KUKA KRL program: MyProgram_278().src

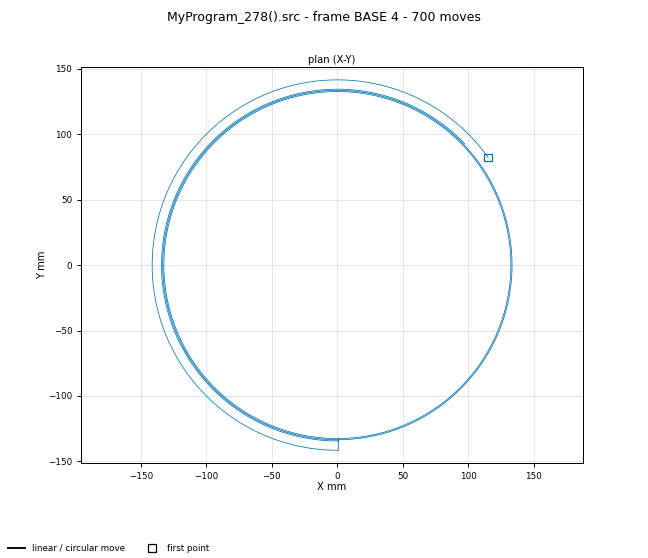
[picture p0: tool path of MyProgram_278().src in frame BASE 4, 700 of 700 moves have a stored position in this frame; points joined in program order, loops and branches not executed]
&ACCESS RVP
&REL 1
&PARAM TEMPLATE = C:\KRC\Roboter\Template\vorgabe
&PARAM EDITMASK = *
DEF MyProgram_278()
; ---- Setting reference (Base) ----
$BASE = BASE_DATA[4]

; --------------------------
; ---- Setting tool (TCP) ----
$TOOL = TOOL_DATA[3]
; --------------------------

$VEL.CP = VEL_APROX_PRINT
Startdeposition()
$VEL.CP = VEL_PRINT
LIN {X 115.1454,Y 82.1588,Z 172,A 37.1025,B 8.4652,C 0.1678,E1 8.5966,E2 414.6408} C_DIS
LIN {X 112.6327,Y 85.5722,Z 172,A 38.7723,B 8.4652,C 0.1649,E1 8.5938,E2 412.9763} C_DIS
LIN {X 109.941,Y 89.0032,Z 172,A 40.5158,B 8.4652,C 0.1614,E1 8.5908,E2 411.2351} C_DIS
LIN {X 107.1131,Y 92.3867,Z 172,A 42.2179,B 8.4653,C 0.1593,E1 8.5877,E2 409.5431} C_DIS
LIN {X 104.5819,Y 95.2429,Z 172,A 43.8363,B 8.4654,C 0.1545,E1 8.5847,E2 407.9148} C_DIS
LIN {X 101.4657,Y 98.556,Z 172,A 45.6031,B 8.4654,C 0.1523,E1 8.5813,E2 406.1572} C_DIS
LIN {X 98.3943,Y 101.6222,Z 172,A 47.3676,B 8.4655,C 0.1486,E1 8.5778,E2 404.3913} C_DIS
LIN {X 95.1433,Y 104.6723,Z 172,A 49.1662,B 8.4655,C 0.1453,E1 8.5741,E2 402.593} C_DIS
LIN {X 91.7276,Y 107.6782,Z 172,A 50.9618,B 8.4656,C 0.1428,E1 8.5703,E2 400.8031} C_DIS
LIN {X 88.3842,Y 110.4395,Z 172,A 52.7089,B 8.4656,C 0.1398,E1 8.5665,E2 399.0569} C_DIS
LIN {X 84.9572,Y 113.0968,Z 172,A 54.4403,B 8.4657,C 0.1373,E1 8.5627,E2 397.3283} C_DIS
LIN {X 81.4292,Y 115.6625,Z 172,A 56.2159,B 8.4657,C 0.1342,E1 8.5587,E2 395.5514} C_DIS
LIN {X 77.8557,Y 118.0975,Z 172,A 57.9483,B 8.4658,C 0.1318,E1 8.5546,E2 393.8213} C_DIS
LIN {X 74.2111,Y 120.4214,Z 172,A 59.7003,B 8.4658,C 0.1291,E1 8.5505,E2 392.069} C_DIS
LIN {X 70.4755,Y 122.6455,Z 172,A 61.4566,B 8.4658,C 0.1267,E1 8.5463,E2 390.3132} C_DIS
LIN {X 66.6565,Y 124.762,Z 172,A 63.2273,B 8.4659,C 0.1242,E1 8.5419,E2 388.5421} C_DIS
LIN {X 62.7995,Y 126.7448,Z 172,A 64.8378,B 8.4659,C 0.1249,E1 8.5379,E2 386.9504} C_DIS
LIN {X 59.6825,Y 128.2423,Z 172,A 66.2482,B 8.4659,C 0.123,E1 8.5344,E2 385.5388} C_DIS
LIN {X 56.3317,Y 129.7488,Z 172,A 67.58,B 8.4659,C 0.1245,E1 8.531,E2 384.2271} C_DIS
LIN {X 53.5262,Y 130.9328,Z 172,A 69.0454,B 8.4659,C 0.1185,E1 8.5272,E2 382.7321} C_DIS
LIN {X 49.8907,Y 132.3593,Z 172,A 70.6218,B 8.466,C 0.117,E1 8.5231,E2 381.1565} C_DIS
LIN {X 46.0135,Y 133.7567,Z 172,A 72.2511,B 8.466,C 0.1162,E1 8.5188,E2 379.5326} C_DIS
LIN {X 41.6859,Y 135.168,Z 172,A 73.8664,B 8.466,C 0.1192,E1 8.5146,E2 377.9469} C_DIS
LIN {X 38.5271,Y 136.1025,Z 172,A 75.2571,B 8.466,C 0.117,E1 8.5108,E2 376.5492} C_DIS
LIN {X 34.9773,Y 137.0571,Z 172,A 76.8136,B 8.466,C 0.1146,E1 8.5066,E2 374.9844} C_DIS
LIN {X 32.0331,Y 137.776,Z 172,A 78.0399,B 8.466,C 0.1138,E1 8.5033,E2 373.7585} C_DIS
LIN {X 28.648,Y 138.5191,Z 172,A 79.439,B 8.466,C 0.1131,E1 8.4994,E2 372.3604} C_DIS
LIN {X 25.2479,Y 139.1787,Z 172,A 80.6426,B 8.466,C 0.1162,E1 8.4962,E2 371.1827} C_DIS
LIN {X 22.4622,Y 139.6574,Z 172,A 81.9857,B 8.466,C 0.1119,E1 8.4924,E2 369.8146} C_DIS
LIN {X 19.0333,Y 140.165,Z 172,A 83.3905,B 8.466,C 0.1113,E1 8.4886,E2 368.4102} C_DIS
LIN {X 15.5815,Y 140.5898,Z 172,A 84.9056,B 8.4661,C 0.1088,E1 8.4843,E2 366.8819} C_DIS
LIN {X 11.0551,Y 141.0194,Z 172,A 86.7804,B 8.4661,C 0.1077,E1 8.4791,E2 365.0036} C_DIS
LIN {X 6.9219,Y 141.2807,Z 172,A 88.3854,B 8.4661,C 0.1089,E1 8.4746,E2 363.4085} C_DIS
LIN {X 2.8123,Y 141.4229,Z 172,A 89.8163,B 8.4661,C 0.1132,E1 8.4707,E2 362.0084} C_DIS
LIN {X -0.0523,Y 141.452,Z 172,A 91.1317,B 8.4661,C 0.1103,E1 8.467,E2 360.6737} C_DIS
LIN {X -3.4727,Y 141.4082,Z 172,A 92.5212,B 8.4661,C 0.1103,E1 8.4631,E2 359.2844} C_DIS
LIN {X -6.9499,Y 141.2793,Z 172,A 93.922,B 8.4661,C 0.1107,E1 8.4592,E2 357.8853} C_DIS
LIN {X -11.0634,Y 141.0188,Z 172,A 95.7118,B 8.4661,C 0.1088,E1 8.4542,E2 356.0811} C_DIS
LIN {X -15.5986,Y 140.588,Z 172,A 97.5605,B 8.4661,C 0.1093,E1 8.4491,E2 354.2329} C_DIS
LIN {X -20.8351,Y 139.9093,Z 172,A 99.5993,B 8.4661,C 0.112,E1 8.4435,E2 352.2082} C_DIS
LIN {X -24.2763,Y 139.3526,Z 172,A 101.0099,B 8.4661,C 0.1128,E1 8.4396,E2 350.7986} C_DIS
LIN {X -27.6797,Y 138.7161,Z 172,A 102.4085,B 8.4661,C 0.1136,E1 8.4357,E2 349.4013} C_DIS
LIN {X -31.0262,Y 138.0059,Z 172,A 103.7935,B 8.4661,C 0.1145,E1 8.432,E2 348.0172} C_DIS
LIN {X -34.3796,Y 137.2088,Z 172,A 105.204,B 8.4661,C 0.1152,E1 8.4281,E2 346.6058} C_DIS
LIN {X -37.7337,Y 136.3243,Z 172,A 106.6143,B 8.4661,C 0.1162,E1 8.4243,E2 345.1958} C_DIS
LIN {X -41.0644,Y 135.3582,Z 172,A 108.0256,B 8.4661,C 0.1173,E1 8.4206,E2 343.7846} C_DIS
LIN {X -44.3704,Y 134.3107,Z 172,A 109.5601,B 8.4661,C 0.1162,E1 8.4164,E2 342.2345} C_DIS
LIN {X -48.2905,Y 132.9516,Z 172,A 111.1286,B 8.466,C 0.1199,E1 8.4124,E2 340.6816} C_DIS
LIN {X -51.531,Y 131.7294,Z 172,A 112.5826,B 8.466,C 0.1205,E1 8.4086,E2 339.2221} C_DIS
LIN {X -55.7331,Y 130.0076,Z 172,A 114.4641,B 8.466,C 0.1218,E1 8.4037,E2 337.3366} C_DIS
LIN {X -59.1861,Y 128.4718,Z 172,A 115.8479,B 8.4659,C 0.1262,E1 8.4002,E2 335.9728} C_DIS
LIN {X -62.0494,Y 127.1148,Z 172,A 117.3081,B 8.4659,C 0.1248,E1 8.3965,E2 334.4911} C_DIS
LIN {X -65.4353,Y 125.4046,Z 172,A 118.8296,B 8.4659,C 0.1271,E1 8.3927,E2 332.9728} C_DIS
LIN {X -69.4478,Y 123.2297,Z 172,A 120.6863,B 8.4659,C 0.1296,E1 8.3882,E2 331.1167} C_DIS
LIN {X -73.1872,Y 121.0461,Z 172,A 122.4642,B 8.4659,C 0.1318,E1 8.3839,E2 329.3372} C_DIS
LIN {X -76.6775,Y 118.8666,Z 172,A 124.2067,B 8.4658,C 0.1331,E1 8.3798,E2 327.5865} C_DIS
LIN {X -80.4753,Y 116.3288,Z 172,A 126.0453,B 8.4658,C 0.1364,E1 8.3756,E2 325.751} C_DIS
LIN {X -84.0458,Y 113.776,Z 172,A 127.823,B 8.4657,C 0.1394,E1 8.3715,E2 323.9749} C_DIS
LIN {X -87.4843,Y 111.1532,Z 172,A 129.5764,B 8.4657,C 0.1425,E1 8.3677,E2 322.2229} C_DIS
LIN {X -90.7455,Y 108.5073,Z 172,A 131.3387,B 8.4656,C 0.1447,E1 8.3639,E2 320.4543} C_DIS
LIN {X -94.1347,Y 105.5807,Z 172,A 133.2066,B 8.4656,C 0.1473,E1 8.3599,E2 318.5812} C_DIS
LIN {X -97.5578,Y 102.4259,Z 172,A 135.0917,B 8.4655,C 0.151,E1 8.3561,E2 316.6979} C_DIS
LIN {X -100.7312,Y 99.307,Z 172,A 136.8846,B 8.4655,C 0.1549,E1 8.3526,E2 314.908} C_DIS
LIN {X -103.7389,Y 96.1607,Z 172,A 138.665,B 8.4654,C 0.1584,E1 8.3491,E2 313.127} C_DIS
LIN {X -106.7016,Y 92.8618,Z 172,A 140.4368,B 8.4653,C 0.1627,E1 8.3459,E2 311.3601} C_DIS
LIN {X -109.1769,Y 89.9391,Z 172,A 142.0776,B 8.4653,C 0.1647,E1 8.3429,E2 309.7093} C_DIS
LIN {X -111.717,Y 86.7632,Z 172,A 143.7599,B 8.4652,C 0.1679,E1 8.34,E2 308.0243} C_DIS
LIN {X -114.3228,Y 83.3004,Z 172,A 145.5562,B 8.4651,C 0.1714,E1 8.337,E2 306.2244} C_DIS
LIN {X -116.9427,Y 79.5804,Z 172,A 147.3892,B 8.4651,C 0.1759,E1 8.3341,E2 304.3946} C_DIS
LIN {X -119.3425,Y 75.9344,Z 172,A 149.1792,B 8.4649,C 0.1799,E1 8.3314,E2 302.6036} C_DIS
LIN {X -121.6068,Y 72.252,Z 172,A 150.9376,B 8.4649,C 0.1842,E1 8.3289,E2 300.846} C_DIS
LIN {X -123.7662,Y 68.487,Z 172,A 152.7274,B 8.4647,C 0.1881,E1 8.3264,E2 299.0539} C_DIS
LIN {X -125.8053,Y 64.6628,Z 172,A 154.5384,B 8.4647,C 0.1917,E1 8.3241,E2 297.2375} C_DIS
LIN {X -127.4923,Y 61.2682,Z 172,A 156.0158,B 8.4646,C 0.1967,E1 8.3223,E2 295.769} C_DIS
LIN {X -128.9555,Y 58.1258,Z 172,A 157.4972,B 8.4645,C 0.1992,E1 8.3205,E2 294.2791} C_DIS
LIN {X -130.4649,Y 54.6526,Z 172,A 158.986,B 8.4644,C 0.204,E1 8.3189,E2 292.7977} C_DIS
LIN {X -131.9767,Y 50.8947,Z 172,A 160.6744,B 8.4643,C 0.2077,E1 8.3172,E2 291.1048} C_DIS
LIN {X -133.1844,Y 47.6449,Z 172,A 162.1014,B 8.4643,C 0.2112,E1 8.3158,E2 289.6764} C_DIS
LIN {X -134.5157,Y 43.7501,Z 172,A 163.9142,B 8.4642,C 0.2134,E1 8.3142,E2 287.8465} C_DIS
LIN {X -135.5481,Y 40.4382,Z 172,A 165.2286,B 8.464,C 0.2188,E1 8.3131,E2 286.5452} C_DIS
LIN {X -136.4988,Y 37.1021,Z 172,A 166.7684,B 8.464,C 0.2206,E1 8.312,E2 284.9894} C_DIS
LIN {X -137.4708,Y 33.3144,Z 172,A 168.1472,B 8.4638,C 0.2283,E1 8.3111,E2 283.6387} C_DIS
LIN {X -138.1673,Y 30.2994,Z 172,A 169.5473,B 8.4638,C 0.2295,E1 8.3102,E2 282.2208} C_DIS
LIN {X -138.8695,Y 26.8965,Z 172,A 170.9776,B 8.4636,C 0.2332,E1 8.3094,E2 280.789} C_DIS
LIN {X -139.3798,Y 24.1242,Z 172,A 172.1369,B 8.4636,C 0.2362,E1 8.3088,E2 279.6286} C_DIS
LIN {X -139.9662,Y 20.4381,Z 172,A 173.5906,B 8.4634,C 0.2414,E1 8.3082,E2 278.1838} C_DIS
LIN {X -140.3869,Y 17.3177,Z 172,A 174.9932,B 8.4634,C 0.2431,E1 8.3077,E2 276.766} C_DIS
LIN {X -140.8329,Y 13.2018,Z 172,A 176.7152,B 8.4632,C 0.2472,E1 8.3072,E2 275.0397} C_DIS
LIN {X -141.1449,Y 9.3056,Z 172,A 178.1959,B 8.4631,C 0.2534,E1 8.3069,E2 273.5738} C_DIS
LIN {X -141.3295,Y 5.8467,Z 172,A 179.5992,B 8.4629,C 0.2574,E1 8.3067,E2 272.1718} C_DIS
LIN {X -141.4227,Y 2.8208,Z 172,A -178.9623,B 8.4629,C 0.2576,E1 8.3067,E2 270.7069} C_DIS
LIN {X -141.4499,Y -0.6582,Z 172,A -177.504,B 8.4629,C 0.2609,E1 8.3067,E2 269.2435} C_DIS
LIN {X -141.3775,Y -4.5742,Z 172,A -175.8333,B 8.4627,C 0.2641,E1 8.3067,E2 267.5633} C_DIS
LIN {X -141.1829,Y -8.6883,Z 172,A -174.2143,B 8.4626,C 0.2697,E1 8.307,E2 265.9522} C_DIS
LIN {X -140.8327,Y -13.2038,Z 172,A -172.3102,B 8.4624,C 0.2739,E1 8.3075,E2 264.0406} C_DIS
LIN {X -140.309,Y -17.9345,Z 172,A -170.4432,B 8.4622,C 0.2804,E1 8.3081,E2 262.1832} C_DIS
LIN {X -139.9212,Y -20.753,Z 172,A -169.2957,B 8.4621,C 0.2838,E1 8.3085,E2 261.0374} C_DIS
LIN {X -139.2931,Y -24.6084,Z 172,A -167.8031,B 8.4619,C 0.2897,E1 8.3092,E2 259.5577} C_DIS
LIN {X -138.7327,Y -27.598,Z 172,A -166.4153,B 8.4619,C 0.2907,E1 8.31,E2 258.1506} C_DIS
LIN {X -138.0138,Y -30.992,Z 172,A -164.988,B 8.4617,C 0.2943,E1 8.3108,E2 256.7216} C_DIS
LIN {X -137.0516,Y -34.9988,Z 172,A -163.2494,B 8.4617,C 0.2978,E1 8.312,E2 254.9751} C_DIS
LIN {X -135.8511,Y -39.4033,Z 172,A -161.4136,B 8.4614,C 0.3031,E1 8.3134,E2 253.1425} C_DIS
LIN {X -134.8446,Y -42.7206,Z 172,A -159.9867,B 8.4614,C 0.3066,E1 8.3146,E2 251.7137} C_DIS
LIN {X -133.5397,Y -46.6396,Z 172,A -158.2855,B 8.4612,C 0.3107,E1 8.3161,E2 250.01} C_DIS
LIN {X -132.2449,Y -50.1963,Z 172,A -156.5727,B 8.4612,C 0.3119,E1 8.3178,E2 248.2747} C_DIS
LIN {X -130.6879,Y -54.1187,Z 172,A -154.9897,B 8.4609,C 0.3185,E1 8.3194,E2 246.7094} C_DIS
LIN {X -129.3124,Y -57.3278,Z 172,A -153.5572,B 8.4607,C 0.3219,E1 8.321,E2 245.2756} C_DIS
LIN {X -127.8683,Y -60.481,Z 172,A -152.1318,B 8.4607,C 0.3251,E1 8.3227,E2 243.8483} C_DIS
LIN {X -126.1996,Y -63.8883,Z 172,A -150.5694,B 8.4605,C 0.3286,E1 8.3247,E2 242.2835} C_DIS
LIN {X -124.5929,Y -66.9712,Z 172,A -149.0497,B 8.4605,C 0.3303,E1 8.3267,E2 240.75} C_DIS
LIN {X -122.3755,Y -70.9421,Z 172,A -147.2166,B 8.4602,C 0.335,E1 8.3292,E2 238.9191} C_DIS
LIN {X -120.1302,Y -74.6812,Z 172,A -145.3688,B 8.4602,C 0.3379,E1 8.3319,E2 237.0616} C_DIS
LIN {X -117.6102,Y -78.59,Z 172,A -143.475,B 8.46,C 0.3422,E1 8.3348,E2 235.1675} C_DIS
LIN {X -115.1466,Y -82.1572,Z 172,A -141.6889,B 8.4598,C 0.3458,E1 8.3377,E2 233.3782} C_DIS
LIN {X -112.5749,Y -85.6478,Z 172,A -139.8928,B 8.4597,C 0.3491,E1 8.3407,E2 231.5777} C_DIS
LIN {X -109.8972,Y -89.0575,Z 172,A -138.0888,B 8.4595,C 0.3521,E1 8.3439,E2 229.7681} C_DIS
LIN {X -107.0913,Y -92.412,Z 172,A -136.3373,B 8.4594,C 0.3562,E1 8.347,E2 228.0199} C_DIS
LIN {X -103.996,Y -95.8822,Z 172,A -134.4237,B 8.4592,C 0.3596,E1 8.3506,E2 226.103} C_DIS
LIN {X -100.8648,Y -99.1708,Z 172,A -132.6103,B 8.4591,C 0.3638,E1 8.3541,E2 224.2937} C_DIS
LIN {X -97.94,Y -102.0605,Z 172,A -130.8665,B 8.459,C 0.3656,E1 8.3576,E2 222.54} C_DIS
LIN {X -94.52,Y -105.2356,Z 172,A -128.9605,B 8.4588,C 0.3689,E1 8.3616,E2 220.6324} C_DIS
LIN {X -91.0669,Y -108.2376,Z 172,A -127.1242,B 8.4587,C 0.3725,E1 8.3655,E2 218.7988} C_DIS
LIN {X -87.7072,Y -110.9782,Z 172,A -125.3297,B 8.4586,C 0.3749,E1 8.3694,E2 216.9996} C_DIS
LIN {X -84.2255,Y -113.6428,Z 172,A -123.5646,B 8.4584,C 0.378,E1 8.3733,E2 215.2362} C_DIS
LIN {X -80.7198,Y -116.1587,Z 172,A -121.8052,B 8.4584,C 0.3806,E1 8.3773,E2 213.4756} C_DIS
LIN {X -77.1326,Y -118.5711,Z 172,A -120.0273,B 8.4582,C 0.3827,E1 8.3815,E2 211.6943} C_DIS
LIN {X -73.4638,Y -120.8789,Z 172,A -118.2109,B 8.4582,C 0.3841,E1 8.3858,E2 209.87} C_DIS
LIN {X -69.6952,Y -123.0906,Z 172,A -116.4181,B 8.4581,C 0.3861,E1 8.3902,E2 208.0743} C_DIS
LIN {X -66.1771,Y -125.0151,Z 172,A -114.9013,B 8.4579,C 0.3901,E1 8.3939,E2 206.5717} C_DIS
LIN {X -62.808,Y -126.7406,Z 172,A -113.3542,B 8.4579,C 0.3917,E1 8.3977,E2 205.0228} C_DIS
LIN {X -59.6948,Y -128.2366,Z 172,A -111.9411,B 8.4578,C 0.393,E1 8.4013,E2 203.6078} C_DIS
LIN {X -56.3261,Y -129.7512,Z 172,A -110.5695,B 8.4576,C 0.3969,E1 8.4048,E2 202.2527} C_DIS
LIN {X -53.5252,Y -130.9332,Z 172,A -109.0853,B 8.4577,C 0.3935,E1 8.4087,E2 200.7348} C_DIS
LIN {X -49.2821,Y -132.5873,Z 172,A -107.3405,B 8.4576,C 0.397,E1 8.4132,E2 199.003} C_DIS
LIN {X -46.0166,Y -133.7557,Z 172,A -105.8454,B 8.4576,C 0.3965,E1 8.4172,E2 197.4957} C_DIS
LIN {X -41.4783,Y -135.2315,Z 172,A -104.0928,B 8.4574,C 0.4014,E1 8.4218,E2 195.7668} C_DIS
LIN {X -38.7552,Y -136.0387,Z 172,A -102.8288,B 8.4574,C 0.4,E1 8.4252,E2 194.4875} C_DIS
LIN {X -34.9861,Y -137.0549,Z 172,A -101.1431,B 8.4574,C 0.399,E1 8.4298,E2 192.7875} C_DIS
LIN {X -30.3504,Y -138.1563,Z 172,A -99.304,B 8.4574,C 0.4018,E1 8.4348,E2 190.96} C_DIS
LIN {X -26.9573,Y -138.8579,Z 172,A -97.8943,B 8.4574,C 0.4023,E1 8.4386,E2 189.5491} C_DIS
LIN {X -24.1772,Y -139.3703,Z 172,A -96.7641,B 8.4573,C 0.403,E1 8.4417,E2 188.4206} C_DIS
LIN {X -20.7465,Y -139.9221,Z 172,A -95.3306,B 8.4573,C 0.403,E1 8.4457,E2 186.9832} C_DIS
LIN {X -17.0562,Y -140.4181,Z 172,A -93.7579,B 8.4573,C 0.4021,E1 8.4501,E2 185.4013} C_DIS
LIN {X -13.2156,Y -140.8316,Z 172,A -92.2298,B 8.4573,C 0.4031,E1 8.4543,E2 183.8775} C_DIS
LIN {X -8.6601,Y -141.1847,Z 172,A -90.418,B 8.4573,C 0.404,E1 8.4594,E2 182.0701} C_DIS
LIN {X -4.5508,Y -141.3782,Z 172,A -88.7312,B 8.4573,C 0.4036,E1 8.4641,E2 180.3799} C_DIS
LIN {X -1.7323,Y -141.4408,Z 172,A -87.6287,B 8.4573,C 0.4043,E1 8.4671,E2 179.2822} C_DIS
LIN {X 1.0226,Y -141.4455,Z 172,A -86.8342,B 8.4569,C 0.4104,E1 8.4692,E2 178.5298} C_DIS
Enddeposition()
LIN {X 0.9597,Y -132.5053,Z 173,A -87.2924,B 8.5827,C 0.3662,E1 8.5925,E2 178.6674} C_DIS
Startdeposition()
$VEL.CP = VEL_PRINT
LIN {X -2.381,Y -132.4898,Z 173,A -88.9158,B 8.5825,C 0.3696,E1 8.5879,E2 180.3133} C_DIS
LIN {X -5.7833,Y -132.3862,Z 173,A -90.3521,B 8.5825,C 0.369,E1 8.5839,E2 181.7461} C_DIS
LIN {X -8.7494,Y -132.2232,Z 173,A -91.7266,B 8.5825,C 0.3706,E1 8.58,E2 183.1321} C_DIS
LIN {X -12.1019,Y -131.9584,Z 173,A -93.3007,B 8.5825,C 0.3725,E1 8.5756,E2 184.7214} C_DIS
LIN {X -16.2246,Y -131.5149,Z 173,A -94.9013,B 8.5825,C 0.3687,E1 8.5712,E2 186.2992} C_DIS
LIN {X -19.4498,Y -131.0776,Z 173,A -96.3155,B 8.5825,C 0.3684,E1 8.5673,E2 187.7147} C_DIS
LIN {X -22.6582,Y -130.5611,Z 173,A -97.7413,B 8.5825,C 0.3684,E1 8.5634,E2 189.1435} C_DIS
LIN {X -25.8503,Y -129.9662,Z 173,A -99.1463,B 8.5826,C 0.3677,E1 8.5595,E2 190.549} C_DIS
LIN {X -29.7453,Y -129.1293,Z 173,A -100.8844,B 8.5826,C 0.3671,E1 8.5548,E2 192.2894} C_DIS
LIN {X -33.7754,Y -128.1345,Z 173,A -102.6831,B 8.5826,C 0.3661,E1 8.5499,E2 194.089} C_DIS
LIN {X -36.9449,Y -127.2566,Z 173,A -104.0949,B 8.5827,C 0.365,E1 8.5461,E2 195.4998} C_DIS
LIN {X -40.4074,Y -126.1995,Z 173,A -105.7344,B 8.5827,C 0.365,E1 8.5417,E2 197.1486} C_DIS
LIN {X -43.8059,Y -125.0611,Z 173,A -107.226,B 8.5828,C 0.3628,E1 8.5378,E2 198.6334} C_DIS
LIN {X -47.0117,Y -123.8922,Z 173,A -108.8671,B 8.5828,C 0.3643,E1 8.5334,E2 200.2948} C_DIS
LIN {X -51.1864,Y -122.2253,Z 173,A -110.7174,B 8.5829,C 0.3608,E1 8.5287,E2 202.1339} C_DIS
LIN {X -54.5147,Y -120.7782,Z 173,A -112.3809,B 8.5829,C 0.3608,E1 8.5244,E2 203.809} C_DIS
LIN {X -58.1203,Y -119.0855,Z 173,A -113.9715,B 8.5831,C 0.3566,E1 8.5204,E2 205.3837} C_DIS
LIN {X -61.0215,Y -117.6258,Z 173,A -115.369,B 8.5831,C 0.3547,E1 8.517,E2 206.7803} C_DIS
LIN {X -63.9076,Y -116.084,Z 173,A -116.9596,B 8.5831,C 0.3559,E1 8.513,E2 208.3922} C_DIS
LIN {X -67.5035,Y -114.0307,Z 173,A -118.6243,B 8.5833,C 0.3514,E1 8.509,E2 210.0417} C_DIS
LIN {X -70.2751,Y -112.3435,Z 173,A -120.0427,B 8.5833,C 0.3496,E1 8.5056,E2 211.4618} C_DIS
LIN {X -73.6197,Y -110.1803,Z 173,A -121.818,B 8.5834,C 0.3479,E1 8.5015,E2 213.2434} C_DIS
LIN {X -77.0465,Y -107.8119,Z 173,A -123.5913,B 8.5836,C 0.3446,E1 8.4974,E2 215.013} C_DIS
LIN {X -79.6565,Y -105.8982,Z 173,A -125.1381,B 8.5836,C 0.3447,E1 8.4939,E2 216.5774} C_DIS
LIN {X -83.0306,Y -103.274,Z 173,A -126.9759,B 8.5836,C 0.3414,E1 8.4899,E2 218.4136} C_DIS
LIN {X -86.277,Y -100.5778,Z 173,A -128.7973,B 8.5838,C 0.3381,E1 8.486,E2 220.2341} C_DIS
LIN {X -89.3334,Y -97.8737,Z 173,A -130.5836,B 8.5839,C 0.3352,E1 8.4823,E2 222.0226} C_DIS
LIN {X -92.2223,Y -95.1557,Z 173,A -132.3094,B 8.5841,C 0.3321,E1 8.4788,E2 223.7492} C_DIS
LIN {X -95.154,Y -92.224,Z 173,A -134.123,B 8.5841,C 0.3288,E1 8.4753,E2 225.5647} C_DIS
LIN {X -97.9916,Y -89.2034,Z 173,A -135.9986,B 8.5843,C 0.3265,E1 8.4717,E2 227.4498} C_DIS
LIN {X -101.1067,Y -85.6565,Z 173,A -138.0254,B 8.5844,C 0.3219,E1 8.468,E2 229.474} C_DIS
LIN {X -103.7467,Y -82.439,Z 173,A -139.8152,B 8.5846,C 0.3178,E1 8.4649,E2 231.262} C_DIS
LIN {X -106.4386,Y -78.9332,Z 173,A -141.8433,B 8.5846,C 0.3153,E1 8.4614,E2 233.3032} C_DIS
LIN {X -108.7586,Y -75.7041,Z 173,A -143.506,B 8.5849,C 0.3105,E1 8.4587,E2 234.9583} C_DIS
LIN {X -111.0758,Y -72.2617,Z 173,A -145.2555,B 8.585,C 0.3056,E1 8.4561,E2 236.7016} C_DIS
LIN {X -113.1978,Y -68.8909,Z 173,A -147.0175,B 8.5852,C 0.302,E1 8.4535,E2 238.4675} C_DIS
LIN {X -114.9544,Y -65.9177,Z 173,A -148.5138,B 8.5852,C 0.2984,E1 8.4513,E2 239.9633} C_DIS
LIN {X -116.8718,Y -62.4551,Z 173,A -150.2717,B 8.5854,C 0.2949,E1 8.449,E2 241.7258} C_DIS
LIN {X -118.3626,Y -59.5793,Z 173,A -151.6868,B 8.5855,C 0.2915,E1 8.4472,E2 243.1417} C_DIS
LIN {X -119.7842,Y -56.6659,Z 173,A -153.1098,B 8.5856,C 0.2883,E1 8.4455,E2 244.5665} C_DIS
LIN {X -121.1428,Y -53.6996,Z 173,A -154.5405,B 8.5857,C 0.2849,E1 8.4438,E2 245.9987} C_DIS
LIN {X -122.4234,Y -50.712,Z 173,A -155.9674,B 8.5858,C 0.2815,E1 8.4423,E2 247.4271} C_DIS
LIN {X -123.9001,Y -46.9905,Z 173,A -157.769,B 8.586,C 0.2779,E1 8.4404,E2 249.236} C_DIS
LIN {X -125.3043,Y -43.1044,Z 173,A -159.5681,B 8.5861,C 0.2733,E1 8.4388,E2 251.0353} C_DIS
LIN {X -126.5848,Y -39.1859,Z 173,A -161.3934,B 8.5862,C 0.2691,E1 8.4372,E2 252.8644} C_DIS
LIN {X -127.5391,Y -35.9575,Z 173,A -162.9581,B 8.5863,C 0.2667,E1 8.436,E2 254.4411} C_DIS
LIN {X -128.7239,Y -31.455,Z 173,A -164.92,B 8.5865,C 0.2603,E1 8.4346,E2 256.3953} C_DIS
LIN {X -129.4826,Y -28.1674,Z 173,A -166.4827,B 8.5865,C 0.2578,E1 8.4337,E2 257.9692} C_DIS
LIN {X -130.2665,Y -24.2924,Z 173,A -168.0949,B 8.5868,C 0.2515,E1 8.4328,E2 259.5685} C_DIS
LIN {X -130.8301,Y -21.0524,Z 173,A -169.5586,B 8.5868,C 0.2481,E1 8.4321,E2 261.036} C_DIS
LIN {X -131.3061,Y -17.8395,Z 173,A -170.9918,B 8.587,C 0.2445,E1 8.4316,E2 262.4715} C_DIS
LIN {X -131.687,Y -14.7654,Z 173,A -172.3999,B 8.587,C 0.2417,E1 8.4311,E2 263.8866} C_DIS
LIN {X -132.0225,Y -11.3691,Z 173,A -173.9578,B 8.5871,C 0.2386,E1 8.4307,E2 265.4529} C_DIS
LIN {X -132.3143,Y -7.2414,Z 173,A -175.6293,B 8.5873,C 0.2317,E1 8.4304,E2 267.109} C_DIS
LIN {X -132.4468,Y -4.1512,Z 173,A -177.0764,B 8.5873,C 0.2295,E1 8.4303,E2 268.5678} C_DIS
LIN {X -132.5145,Y 0.0019,Z 173,A -179.0708,B 8.5874,C 0.2272,E1 8.4303,E2 270.5841} C_DIS
LIN {X -132.4471,Y 4.1413,Z 173,A 179.3434,B 8.5877,C 0.219,E1 8.4303,E2 272.1441} C_DIS
LIN {X -132.3149,Y 7.2293,Z 173,A 177.943,B 8.5877,C 0.2161,E1 8.4305,E2 273.5508} C_DIS
LIN {X -132.0346,Y 11.2266,Z 173,A 176.1471,B 8.5878,C 0.212,E1 8.4309,E2 275.3525} C_DIS
LIN {X -131.6023,Y 15.4923,Z 173,A 174.1997,B 8.5879,C 0.208,E1 8.4315,E2 277.3092} C_DIS
LIN {X -131.0789,Y 19.4409,Z 173,A 172.5751,B 8.5881,C 0.2016,E1 8.4321,E2 278.9207} C_DIS
LIN {X -130.5949,Y 22.4616,Z 173,A 171.2403,B 8.5881,C 0.198,E1 8.4327,E2 280.2556} C_DIS
LIN {X -129.9526,Y 25.9171,Z 173,A 169.687,B 8.5882,C 0.1942,E1 8.4336,E2 281.8114} C_DIS
LIN {X -129.1237,Y 29.7699,Z 173,A 167.9225,B 8.5883,C 0.1902,E1 8.4346,E2 283.5813} C_DIS
LIN {X -128.133,Y 33.7809,Z 173,A 166.1187,B 8.5884,C 0.1854,E1 8.4359,E2 285.3854} C_DIS
LIN {X -127.06,Y 37.6163,Z 173,A 164.3416,B 8.5885,C 0.1814,E1 8.4372,E2 287.1672} C_DIS
LIN {X -125.8238,Y 41.5635,Z 173,A 162.5506,B 8.5886,C 0.1765,E1 8.4388,E2 288.9568} C_DIS
LIN {X -124.5199,Y 45.3211,Z 173,A 160.7496,B 8.5886,C 0.173,E1 8.4404,E2 290.7656} C_DIS
LIN {X -123.037,Y 49.2044,Z 173,A 158.904,B 8.5888,C 0.1688,E1 8.4423,E2 292.615} C_DIS
LIN {X -121.4322,Y 53.0424,Z 173,A 157.1426,B 8.5888,C 0.1634,E1 8.4442,E2 294.3702} C_DIS
LIN {X -119.7861,Y 56.6619,Z 173,A 155.405,B 8.589,C 0.1592,E1 8.4463,E2 296.1083} C_DIS
LIN {X -118.3617,Y 59.581,Z 173,A 153.9803,B 8.589,C 0.1558,E1 8.448,E2 297.534} C_DIS
LIN {X -116.867,Y 62.464,Z 173,A 152.5289,B 8.589,C 0.1529,E1 8.4499,E2 298.9895} C_DIS
LIN {X -114.8994,Y 66.0141,Z 173,A 150.7336,B 8.5891,C 0.149,E1 8.4524,E2 300.7878} C_DIS
LIN {X -113.1833,Y 68.9149,Z 173,A 149.2803,B 8.5892,C 0.1453,E1 8.4545,E2 302.2391} C_DIS
LIN {X -111.473,Y 71.6476,Z 173,A 147.868,B 8.5892,C 0.1421,E1 8.4566,E2 303.6522} C_DIS
LIN {X -109.2807,Y 74.9485,Z 173,A 145.9887,B 8.5892,C 0.1405,E1 8.4595,E2 305.5491} C_DIS
LIN {X -106.8723,Y 78.3446,Z 173,A 144.3089,B 8.5894,C 0.1344,E1 8.4623,E2 307.213} C_DIS
LIN {X -104.4711,Y 81.52,Z 173,A 142.4663,B 8.5894,C 0.1322,E1 8.4654,E2 309.0681} C_DIS
LIN {X -101.91,Y 84.6992,Z 173,A 140.684,B 8.5894,C 0.1285,E1 8.4686,E2 310.8507} C_DIS
LIN {X -99.0269,Y 88.0532,Z 173,A 138.7326,B 8.5895,C 0.1249,E1 8.4722,E2 312.8048} C_DIS
LIN {X -96.2776,Y 91.0505,Z 173,A 136.9714,B 8.5895,C 0.1212,E1 8.4755,E2 314.5646} C_DIS
LIN {X -93.3768,Y 94.023,Z 173,A 135.1693,B 8.5896,C 0.1175,E1 8.479,E2 316.3657} C_DIS
LIN {X -90.4564,Y 96.8361,Z 173,A 133.3818,B 8.5896,C 0.1145,E1 8.4827,E2 318.1556} C_DIS
LIN {X -87.4521,Y 99.5583,Z 173,A 131.5938,B 8.5897,C 0.1116,E1 8.4864,E2 319.946} C_DIS
LIN {X -84.3407,Y 102.2069,Z 173,A 129.8318,B 8.5897,C 0.1082,E1 8.4902,E2 321.7058} C_DIS
LIN {X -81.2337,Y 104.6931,Z 173,A 128.0528,B 8.5897,C 0.106,E1 8.4941,E2 323.49} C_DIS
LIN {X -78.6888,Y 106.6195,Z 173,A 126.6434,B 8.5898,C 0.1041,E1 8.4972,E2 324.9016} C_DIS
LIN {X -75.4206,Y 108.9559,Z 173,A 124.8966,B 8.5898,C 0.1013,E1 8.5012,E2 326.648} C_DIS
LIN {X -72.2432,Y 111.0878,Z 173,A 123.3388,B 8.5898,C 0.0971,E1 8.5048,E2 328.193} C_DIS
LIN {X -69.501,Y 112.8239,Z 173,A 121.7857,B 8.5898,C 0.0973,E1 8.5085,E2 329.7624} C_DIS
LIN {X -65.9466,Y 114.9379,Z 173,A 120.1216,B 8.5899,C 0.0927,E1 8.5125,E2 331.4105} C_DIS
LIN {X -62.4687,Y 116.8645,Z 173,A 118.3572,B 8.5899,C 0.091,E1 8.5169,E2 333.1788} C_DIS
LIN {X -59.5869,Y 118.3587,Z 173,A 116.9597,B 8.5899,C 0.089,E1 8.5203,E2 334.5744} C_DIS
LIN {X -56.6527,Y 119.7905,Z 173,A 115.5396,B 8.5899,C 0.0874,E1 8.5239,E2 335.9943} C_DIS
LIN {X -53.6996,Y 121.1428,Z 173,A 114.1226,B 8.59,C 0.0859,E1 8.5275,E2 337.4117} C_DIS
LIN {X -50.6793,Y 122.437,Z 173,A 112.6975,B 8.59,C 0.0843,E1 8.5312,E2 338.8362} C_DIS
LIN {X -47.6723,Y 123.6387,Z 173,A 111.2891,B 8.59,C 0.0829,E1 8.5348,E2 340.2445} C_DIS
LIN {X -44.6334,Y 124.7679,Z 173,A 109.7555,B 8.59,C 0.0837,E1 8.5389,E2 341.7925} C_DIS
LIN {X -40.8715,Y 126.0512,Z 173,A 108.1051,B 8.59,C 0.081,E1 8.5432,E2 343.4337} C_DIS
LIN {X -37.6298,Y 127.0561,Z 173,A 106.6764,B 8.59,C 0.0791,E1 8.5471,E2 344.8568} C_DIS
LIN {X -33.7713,Y 128.1356,Z 173,A 104.7966,B 8.59,C 0.0802,E1 8.5522,E2 346.7526} C_DIS
LIN {X -29.5409,Y 129.176,Z 173,A 102.9667,B 8.59,C 0.078,E1 8.5571,E2 348.575} C_DIS
LIN {X -25.8433,Y 129.9676,Z 173,A 101.4112,B 8.59,C 0.0757,E1 8.5613,E2 350.1203} C_DIS
LIN {X -22.6485,Y 130.5629,Z 173,A 100.0051,B 8.5901,C 0.0749,E1 8.5652,E2 351.5257} C_DIS
LIN {X -19.4417,Y 131.0788,Z 173,A 98.5726,B 8.5901,C 0.0748,E1 8.5692,E2 352.9606} C_DIS
LIN {X -16.2228,Y 131.5152,Z 173,A 97.164,B 8.5901,C 0.0743,E1 8.5731,E2 354.3688} C_DIS
LIN {X -12.9861,Y 131.8735,Z 173,A 95.7576,B 8.5901,C 0.0738,E1 8.577,E2 355.7743} C_DIS
LIN {X -9.4578,Y 132.1732,Z 173,A 94.1414,B 8.5901,C 0.0749,E1 8.5815,E2 357.3996} C_DIS
LIN {X -5.766,Y 132.3869,Z 173,A 92.6148,B 8.5901,C 0.0734,E1 8.5857,E2 358.917} C_DIS
LIN {X -2.2547,Y 132.4919,Z 173,A 91.0315,B 8.5901,C 0.0744,E1 8.5902,E2 360.5071} C_DIS
LIN {X 1.6374,Y 132.5022,Z 173,A 89.4118,B 8.5901,C 0.0733,E1 8.5947,E2 362.1187} C_DIS
LIN {X 4.8828,Y 132.4213,Z 173,A 88.0191,B 8.5901,C 0.0732,E1 8.5985,E2 363.5095} C_DIS
LIN {X 8.3922,Y 132.2452,Z 173,A 86.4048,B 8.5901,C 0.0751,E1 8.6031,E2 365.1342} C_DIS
LIN {X 12.0962,Y 131.9589,Z 173,A 84.8459,B 8.5901,C 0.0746,E1 8.6074,E2 366.6871} C_DIS
LIN {X 16.2274,Y 131.5146,Z 173,A 83.1228,B 8.5901,C 0.0739,E1 8.6122,E2 368.4009} C_DIS
LIN {X 19.4474,Y 131.078,Z 173,A 81.7178,B 8.5901,C 0.0744,E1 8.616,E2 369.8056} C_DIS
LIN {X 22.6549,Y 130.5617,Z 173,A 80.2978,B 8.5901,C 0.0753,E1 8.62,E2 371.2269} C_DIS
LIN {X 25.8477,Y 129.9667,Z 173,A 78.9007,B 8.5901,C 0.0759,E1 8.6238,E2 372.6227} C_DIS
LIN {X 29.755,Y 129.1271,Z 173,A 77.1616,B 8.5901,C 0.0772,E1 8.6285,E2 374.3627} C_DIS
LIN {X 33.8136,Y 128.1243,Z 173,A 75.3866,B 8.5901,C 0.0778,E1 8.6333,E2 376.1335} C_DIS
LIN {X 36.9278,Y 127.2616,Z 173,A 73.9955,B 8.5901,C 0.0788,E1 8.6371,E2 377.5236} C_DIS
LIN {X 40.8724,Y 126.051,Z 173,A 72.2206,B 8.5901,C 0.0802,E1 8.6418,E2 379.2971} C_DIS
LIN {X 44.646,Y 124.7633,Z 173,A 70.3505,B 8.5901,C 0.0845,E1 8.6468,E2 381.184} C_DIS
LIN {X 49.2064,Y 123.0362,Z 173,A 68.3019,B 8.5901,C 0.0855,E1 8.6521,E2 383.2254} C_DIS
LIN {X 53.0254,Y 121.4396,Z 173,A 66.6277,B 8.5901,C 0.0854,E1 8.6563,E2 384.886} C_DIS
LIN {X 56.6534,Y 119.7902,Z 173,A 64.9264,B 8.59,C 0.087,E1 8.6606,E2 386.5847} C_DIS
LIN {X 59.5734,Y 118.3656,Z 173,A 63.604,B 8.59,C 0.0872,E1 8.6639,E2 387.8974} C_DIS
LIN {X 62.4779,Y 116.8595,Z 173,A 62.1271,B 8.59,C 0.0903,E1 8.6676,E2 389.3817} C_DIS
LIN {X 65.9613,Y 114.9295,Z 173,A 60.3896,B 8.59,C 0.093,E1 8.6718,E2 391.1211} C_DIS
LIN {X 69.5154,Y 112.8151,Z 173,A 58.639,B 8.59,C 0.0949,E1 8.676,E2 392.8675} C_DIS
LIN {X 72.399,Y 110.9866,Z 173,A 57.0259,B 8.5899,C 0.0998,E1 8.6798,E2 394.4968} C_DIS
LIN {X 75.7245,Y 108.7445,Z 173,A 55.4111,B 8.5899,C 0.1003,E1 8.6835,E2 396.0977} C_DIS
LIN {X 78.9333,Y 106.4385,Z 173,A 53.6782,B 8.5899,C 0.1037,E1 8.6874,E2 397.8338} C_DIS
LIN {X 82.1697,Y 103.9608,Z 173,A 51.9435,B 8.5898,C 0.1062,E1 8.6913,E2 399.5656} C_DIS
LIN {X 85.3168,Y 101.3934,Z 173,A 50.1759,B 8.5898,C 0.1097,E1 8.6951,E2 401.335} C_DIS
LIN {X 88.6954,Y 98.4522,Z 173,A 48.2852,B 8.5897,C 0.1124,E1 8.699,E2 403.2207} C_DIS
LIN {X 91.641,Y 95.7158,Z 173,A 46.5831,B 8.5897,C 0.1151,E1 8.7025,E2 404.919} C_DIS
LIN {X 94.9019,Y 92.4844,Z 173,A 44.6063,B 8.5897,C 0.119,E1 8.7064,E2 406.8955} C_DIS
LIN {X 97.8877,Y 89.318,Z 173,A 42.7388,B 8.5896,C 0.1227,E1 8.7099,E2 408.762} C_DIS
LIN {X 100.637,Y 86.2083,Z 173,A 40.9771,B 8.5896,C 0.1259,E1 8.7131,E2 410.5205} C_DIS
LIN {X 103.2502,Y 83.0601,Z 173,A 39.2651,B 8.5895,C 0.1287,E1 8.7161,E2 412.2264} C_DIS
LIN {X 105.9051,Y 79.6474,Z 173,A 37.4149,B 8.5895,C 0.1325,E1 8.7193,E2 414.0751} C_DIS
LIN {X 108.3441,Y 76.2963,Z 173,A 35.7052,B 8.5894,C 0.135,E1 8.7221,E2 415.7759} C_DIS
LIN {X 110.1816,Y 73.6178,Z 173,A 34.3229,B 8.5894,C 0.1379,E1 8.7242,E2 417.1562} C_DIS
LIN {X 111.9531,Y 70.895,Z 173,A 32.9405,B 8.5893,C 0.1409,E1 8.7263,E2 418.5367} C_DIS
LIN {X 114.0319,Y 67.5014,Z 173,A 31.2081,B 8.5893,C 0.1453,E1 8.7288,E2 420.2714} C_DIS
LIN {X 115.7271,Y 64.552,Z 173,A 29.6438,B 8.5891,C 0.1509,E1 8.731,E2 421.8477} C_DIS
LIN {X 117.3482,Y 61.5501,Z 173,A 28.2565,B 8.5891,C 0.1528,E1 8.7328,E2 423.2253} C_DIS
LIN {X 119.0863,Y 58.1189,Z 173,A 26.6952,B 8.5891,C 0.155,E1 8.7347,E2 424.7756} C_DIS
LIN {X 120.4747,Y 55.1824,Z 173,A 25.3137,B 8.589,C 0.1582,E1 8.7363,E2 426.1552} C_DIS
LIN {X 121.7437,Y 52.322,Z 173,A 23.9687,B 8.589,C 0.1616,E1 8.7378,E2 427.5001} C_DIS
LIN {X 123.0479,Y 49.1774,Z 173,A 22.4078,B 8.5888,C 0.1674,E1 8.7395,E2 429.0726} C_DIS
LIN {X 124.7672,Y 44.6352,Z 173,A 20.47,B 8.5888,C 0.1697,E1 8.7413,E2 430.9925} C_DIS
LIN {X 125.8213,Y 41.571,Z 173,A 19.0922,B 8.5887,C 0.173,E1 8.7426,E2 432.3685} C_DIS
LIN {X 126.9564,Y 37.9701,Z 173,A 17.3724,B 8.5886,C 0.1794,E1 8.744,E2 434.1} C_DIS
LIN {X 127.9453,Y 34.4847,Z 173,A 15.9422,B 8.5886,C 0.1809,E1 8.7451,E2 435.5151} C_DIS
LIN {X 128.7534,Y 31.3325,Z 173,A 14.4324,B 8.5884,C 0.1869,E1 8.7461,E2 437.0382} C_DIS
LIN {X 129.639,Y 27.4432,Z 173,A 12.8703,B 8.5884,C 0.1884,E1 8.747,E2 438.5822} C_DIS
LIN {X 130.2736,Y 24.2553,Z 173,A 11.4916,B 8.5883,C 0.1918,E1 8.7477,E2 439.9588} C_DIS
LIN {X 130.8297,Y 21.0545,Z 173,A 10.115,B 8.5883,C 0.1953,E1 8.7484,E2 441.3333} C_DIS
LIN {X 131.3081,Y 17.8241,Z 173,A 8.7008,B 8.5881,C 0.1993,E1 8.7489,E2 442.7489} C_DIS
LIN {X 131.7047,Y 14.6014,Z 173,A 7.174,B 8.588,C 0.2059,E1 8.7494,E2 444.2916} C_DIS
LIN {X 132.0843,Y 10.6376,Z 173,A 5.6553,B 8.588,C 0.2066,E1 8.7498,E2 445.7874} C_DIS
LIN {X 132.3142,Y 7.2437,Z 173,A 4.2179,B 8.5879,C 0.2102,E1 8.75,E2 447.2221} C_DIS
LIN {X 132.4474,Y 4.1308,Z 173,A 2.8212,B 8.5878,C 0.2151,E1 8.7502,E2 448.626} C_DIS
LIN {X 132.5145,Y -0.0034,Z 173,A 0.9018,B 8.5876,C 0.2231,E1 8.7502,E2 450.5629} C_DIS
LIN {X 132.4472,Y -4.1388,Z 173,A -0.6298,B 8.5876,C 0.2228,E1 8.7502,E2 452.0651} C_DIS
LIN {X 132.3265,Y -6.9997,Z 173,A -1.912,B 8.5874,C 0.2274,E1 8.75,E2 453.3538} C_DIS
LIN {X 132.0915,Y -10.5521,Z 173,A -3.3716,B 8.5874,C 0.2301,E1 8.7497,E2 454.8053} C_DIS
LIN {X 131.7853,Y -13.8521,Z 173,A -4.7988,B 8.5873,C 0.2342,E1 8.7493,E2 456.2331} C_DIS
LIN {X 131.3072,Y -17.831,Z 173,A -6.4768,B 8.5872,C 0.238,E1 8.7487,E2 457.9062} C_DIS
LIN {X 130.8319,Y -21.0414,Z 173,A -7.8554,B 8.5871,C 0.2415,E1 8.7481,E2 459.2833} C_DIS
LIN {X 130.1349,Y -24.9805,Z 173,A -9.5679,B 8.5869,C 0.2461,E1 8.7472,E2 460.9953} C_DIS
LIN {X 129.442,Y -28.3554,Z 173,A -11.1838,B 8.5867,C 0.253,E1 8.7463,E2 462.628} C_DIS
LIN {X 128.5264,Y -32.252,Z 173,A -12.872,B 8.5867,C 0.257,E1 8.7452,E2 464.3127} C_DIS
LIN {X 127.2828,Y -36.8554,Z 173,A -14.9135,B 8.5864,C 0.2624,E1 8.7436,E2 466.3538} C_DIS
LIN {X 125.9448,Y -41.2002,Z 173,A -16.8095,B 8.5864,C 0.2664,E1 8.742,E2 468.2434} C_DIS
LIN {X 124.5129,Y -45.3406,Z 173,A -18.576,B 8.5862,C 0.269,E1 8.7404,E2 469.9963} C_DIS
LIN {X 123.0368,Y -49.2049,Z 173,A -20.393,B 8.5861,C 0.2745,E1 8.7386,E2 471.8186} C_DIS
LIN {X 121.4128,Y -53.0873,Z 173,A -22.1152,B 8.586,C 0.2773,E1 8.7367,E2 473.5309} C_DIS
LIN {X 120.1518,Y -55.8807,Z 173,A -23.418,B 8.5859,C 0.2804,E1 8.7352,E2 474.8323} C_DIS
LIN {X 118.4682,Y -59.3719,Z 173,A -25.1395,B 8.5857,C 0.2858,E1 8.733,E2 476.5611} C_DIS
LIN {X 116.8681,Y -62.4619,Z 173,A -26.5418,B 8.5857,C 0.2876,E1 8.7312,E2 477.9525} C_DIS
LIN {X 114.9503,Y -65.9249,Z 173,A -28.2622,B 8.5855,C 0.2922,E1 8.7289,E2 479.6757} C_DIS
LIN {X 113.2023,Y -68.8836,Z 173,A -29.8448,B 8.5853,C 0.2979,E1 8.7266,E2 481.2716} C_DIS
LIN {X 110.7799,Y -72.7145,Z 173,A -31.7021,B 8.5853,C 0.3007,E1 8.7238,E2 483.1184} C_DIS
LIN {X 108.8022,Y -75.6415,Z 173,A -33.1491,B 8.5851,C 0.3028,E1 8.7215,E2 484.5573} C_DIS
LIN {X 106.8711,Y -78.3462,Z 173,A -34.5455,B 8.5851,C 0.3054,E1 8.7192,E2 485.9502} C_DIS
LIN {X 104.9621,Y -80.8867,Z 173,A -35.9877,B 8.5849,C 0.3101,E1 8.7168,E2 487.4021} C_DIS
LIN {X 102.3196,Y -84.2047,Z 173,A -37.7965,B 8.5847,C 0.3138,E1 8.7136,E2 489.2097} C_DIS
LIN {X 99.5407,Y -87.4721,Z 173,A -39.635,B 8.5846,C 0.3176,E1 8.7103,E2 491.048} C_DIS
LIN {X 96.8313,Y -90.4616,Z 173,A -41.3469,B 8.5845,C 0.3208,E1 8.707,E2 492.7577} C_DIS
LIN {X 94.0148,Y -93.3851,Z 173,A -43.1064,B 8.5843,C 0.3247,E1 8.7036,E2 494.5194} C_DIS
LIN {X 90.9932,Y -96.3317,Z 173,A -44.8594,B 8.5843,C 0.327,E1 8.7001,E2 496.2654} C_DIS
LIN {X 88.0485,Y -99.0311,Z 173,A -46.5906,B 8.5841,C 0.3306,E1 8.6965,E2 497.9988} C_DIS
LIN {X 84.9737,Y -101.6814,Z 173,A -48.318,B 8.584,C 0.3335,E1 8.6928,E2 499.7245} C_DIS
LIN {X 81.7995,Y -104.2516,Z 173,A -50.0471,B 8.5839,C 0.3361,E1 8.689,E2 501.4507} C_DIS
LIN {X 78.348,Y -106.8698,Z 173,A -51.9757,B 8.5837,C 0.3406,E1 8.6847,E2 503.3879} C_DIS
LIN {X 74.9651,Y -109.2694,Z 173,A -53.763,B 8.5837,C 0.3436,E1 8.6806,E2 505.1761} C_DIS
LIN {X 70.9752,Y -111.9025,Z 173,A -55.7074,B 8.5836,C 0.3446,E1 8.6761,E2 507.1074} C_DIS
LIN {X 67.4216,Y -114.079,Z 173,A -57.4779,B 8.5835,C 0.3469,E1 8.6719,E2 508.8756} C_DIS
LIN {X 64.5322,Y -115.7381,Z 173,A -59.0217,B 8.5833,C 0.3511,E1 8.6681,E2 510.4333} C_DIS
LIN {X 61.0316,Y -117.6205,Z 173,A -60.588,B 8.5833,C 0.3506,E1 8.6642,E2 511.9824} C_DIS
LIN {X 58.1127,Y -119.0893,Z 173,A -61.9865,B 8.5833,C 0.3523,E1 8.6607,E2 513.3803} C_DIS
LIN {X 55.1766,Y -120.4774,Z 173,A -63.5155,B 8.5831,C 0.3566,E1 8.6568,E2 514.9256} C_DIS
LIN {X 50.9423,Y -122.3272,Z 173,A -65.3941,B 8.5831,C 0.3568,E1 8.652,E2 516.7913} C_DIS
LIN {X 47.01,Y -123.8928,Z 173,A -67.2197,B 8.583,C 0.3588,E1 8.6473,E2 518.6178} C_DIS
LIN {X 43.21,Y -125.2677,Z 173,A -68.9409,B 8.583,C 0.3602,E1 8.6428,E2 520.3371} C_DIS
LIN {X 39.4883,Y -126.4923,Z 173,A -70.7013,B 8.5828,C 0.3632,E1 8.6381,E2 522.1068} C_DIS
LIN {X 36.0403,Y -127.5159,Z 173,A -72.2805,B 8.5828,C 0.365,E1 8.6338,E2 523.6901} C_DIS
LIN {X 31.4798,Y -128.7179,Z 173,A -74.2146,B 8.5828,C 0.3647,E1 8.6286,E2 525.6127} C_DIS
LIN {X 27.4453,Y -129.6385,Z 173,A -75.9471,B 8.5828,C 0.365,E1 8.6239,E2 527.3395} C_DIS
LIN {X 24.2397,Y -130.2765,Z 173,A -77.35,B 8.5827,C 0.3658,E1 8.62,E2 528.7421} C_DIS
LIN {X 21.0402,Y -130.8321,Z 173,A -78.7719,B 8.5827,C 0.3669,E1 8.6161,E2 530.1669} C_DIS
LIN {X 17.8294,Y -131.3074,Z 173,A -80.3266,B 8.5825,C 0.3705,E1 8.6118,E2 531.741} C_DIS
LIN {X 13.4826,Y -131.8251,Z 173,A -82.1822,B 8.5825,C 0.3706,E1 8.6066,E2 533.5931} C_DIS
LIN {X 9.4726,Y -132.1721,Z 173,A -83.8789,B 8.5825,C 0.3704,E1 8.6019,E2 535.2854} C_DIS
LIN {X 5.2054,Y -132.4088,Z 173,A -85.6735,B 8.5825,C 0.3699,E1 8.5969,E2 537.0745} C_DIS
LIN {X 1.6252,Y -132.5024,Z 173,A -87.2609,B 8.5825,C 0.3709,E1 8.5925,E2 538.6674} C_DIS
LIN {X 1.6252,Y -132.5024,Z 173,A -87.2609,B 8.5825,C 0.3709,E1 8.5925,E2 538.6674} C_DIS
Enddeposition()
LIN {X 0.9681,Y -133.4137,Z 173,A -87.0186,B 8.5826,C 0.3663,E1 8.5932,E2 538.3942} C_DIS
Startdeposition()
$VEL.CP = VEL_PRINT
LIN {X 4.2482,Y -133.353,Z 173,A -85.2742,B 8.5829,C 0.3598,E1 8.5982,E2 536.6075} C_DIS
LIN {X 8.8754,Y -133.1257,Z 173,A -83.3619,B 8.5829,C 0.3606,E1 8.6035,E2 534.7038} C_DIS
LIN {X 11.9152,Y -132.8882,Z 173,A -81.9972,B 8.5829,C 0.3591,E1 8.6073,E2 533.3315} C_DIS
LIN {X 15.528,Y -132.513,Z 173,A -80.4978,B 8.5829,C 0.3596,E1 8.6115,E2 531.8387} C_DIS
LIN {X 19.2223,Y -132.0279,Z 173,A -78.927,B 8.5829,C 0.3593,E1 8.6158,E2 530.2706} C_DIS
LIN {X 23.1,Y -131.405,Z 173,A -77.2266,B 8.5829,C 0.358,E1 8.6205,E2 528.5675} C_DIS
LIN {X 26.6135,Y -130.738,Z 173,A -75.7586,B 8.5829,C 0.3583,E1 8.6245,E2 527.1069} C_DIS
LIN {X 29.9177,Y -130.0218,Z 173,A -74.2638,B 8.5831,C 0.3564,E1 8.6286,E2 525.6057} C_DIS
LIN {X 34.0105,Y -129.0121,Z 173,A -72.4766,B 8.5831,C 0.3553,E1 8.6334,E2 523.8202} C_DIS
LIN {X 37.2231,Y -128.1218,Z 173,A -71.0217,B 8.5831,C 0.3536,E1 8.6373,E2 522.3614} C_DIS
LIN {X 40.4998,Y -127.1238,Z 173,A -69.8,B 8.5831,C 0.357,E1 8.6405,E2 521.1697} C_DIS
LIN {X 42.6455,Y -126.4211,Z 173,A -68.2915,B 8.5835,C 0.3454,E1 8.6447,E2 519.5932} C_DIS
LIN {X 46.0531,Y -125.2214,Z 173,A -66.9798,B 8.5834,C 0.3484,E1 8.6481,E2 518.3105} C_DIS
LIN {X 49.8004,Y -123.7763,Z 173,A -65.3357,B 8.5834,C 0.348,E1 8.6523,E2 516.675} C_DIS
LIN {X 53.3713,Y -122.2798,Z 173,A -63.6865,B 8.5834,C 0.3462,E1 8.6565,E2 515.0262} C_DIS
LIN {X 57.1603,Y -120.5549,Z 173,A -61.9098,B 8.5836,C 0.344,E1 8.661,E2 513.2493} C_DIS
LIN {X 62.3235,Y -117.9683,Z 173,A -58.8216,B 8.5842,C 0.3282,E1 8.6689,E2 510.0829} C_DIS
LIN {X 67.0153,Y -115.3696,Z 173,A -56.716,B 8.5842,C 0.3287,E1 8.6739,E2 508.0002} C_DIS
LIN {X 70.7411,Y -113.1236,Z 173,A -55.248,B 8.584,C 0.3338,E1 8.6773,E2 506.5807} C_DIS
LIN {X 74.5435,Y -110.655,Z 173,A -53.3169,B 8.584,C 0.3308,E1 8.6818,E2 504.6498} C_DIS
LIN {X 78.5542,Y -107.8448,Z 173,A -51.2729,B 8.5842,C 0.3283,E1 8.6864,E2 502.6113} C_DIS
LIN {X 81.1632,Y -105.8948,Z 173,A -49.5453,B 8.5845,C 0.3189,E1 8.6904,E2 500.8412} C_DIS
LIN {X 84.275,Y -103.4356,Z 173,A -48.1976,B 8.5844,C 0.323,E1 8.6932,E2 499.5365} C_DIS
LIN {X 87.4652,Y -100.7528,Z 173,A -46.3894,B 8.5845,C 0.3191,E1 8.697,E2 497.7243} C_DIS
LIN {X 90.4147,Y -98.1141,Z 173,A -44.9439,B 8.5845,C 0.3209,E1 8.7,E2 496.3088} C_DIS
LIN {X 94.4893,Y -94.1965,Z 173,A -42.3475,B 8.5848,C 0.3124,E1 8.7052,E2 493.689} C_DIS
LIN {X 97.5396,Y -91.0342,Z 173,A -40.4815,B 8.5848,C 0.3087,E1 8.7088,E2 491.8237} C_DIS
LIN {X 100.2247,Y -88.0698,Z 173,A -38.2912,B 8.5854,C 0.2949,E1 8.713,E2 489.5727} C_DIS
LIN {X 103.3408,Y -84.391,Z 173,A -36.7548,B 8.5852,C 0.3014,E1 8.7156,E2 488.101} C_DIS
LIN {X 105.7583,Y -81.3417,Z 173,A -35.0855,B 8.5852,C 0.2975,E1 8.7184,E2 486.4302} C_DIS
LIN {X 108.3387,Y -77.8718,Z 173,A -33.3157,B 8.5854,C 0.2949,E1 8.7213,E2 484.6694} C_DIS
LIN {X 111.2182,Y -73.7011,Z 173,A -31.0845,B 8.5856,C 0.2884,E1 8.7248,E2 482.4291} C_DIS
LIN {X 113.4565,Y -70.2062,Z 173,A -29.3935,B 8.5856,C 0.2859,E1 8.7273,E2 480.7477} C_DIS
LIN {X 115.1802,Y -67.3406,Z 173,A -27.5859,B 8.5861,C 0.2743,E1 8.73,E2 478.8923} C_DIS
LIN {X 117.212,Y -63.7382,Z 173,A -26.2071,B 8.5859,C 0.2782,E1 8.7317,E2 477.5612} C_DIS
LIN {X 118.8619,Y -60.6009,Z 173,A -24.8724,B 8.5859,C 0.2782,E1 8.7334,E2 476.2481} C_DIS
LIN {X 120.9747,Y -56.2658,Z 173,A -22.2554,B 8.5865,C 0.261,E1 8.7366,E2 473.5611} C_DIS
LIN {X 122.8065,Y -52.1521,Z 173,A -20.7481,B 8.5863,C 0.2649,E1 8.7382,E2 472.1051} C_DIS
LIN {X 124.2865,Y -48.5133,Z 173,A -19.1482,B 8.5864,C 0.2622,E1 8.7399,E2 470.5141} C_DIS
LIN {X 125.5276,Y -45.2049,Z 173,A -17.812,B 8.5864,C 0.2619,E1 8.7412,E2 469.1987} C_DIS
LIN {X 127.4104,Y -39.5929,Z 173,A -15.3051,B 8.5866,C 0.2556,E1 8.7434,E2 466.6937} C_DIS
LIN {X 129.3266,Y -32.792,Z 173,A -11.8133,B 8.5872,C 0.2372,E1 8.746,E2 463.1424} C_DIS
LIN {X 130.2532,Y -28.9032,Z 173,A -10.3945,B 8.5872,C 0.2388,E1 8.7468,E2 461.7588} C_DIS
LIN {X 131.0698,Y -24.9285,Z 173,A -8.7954,B 8.5872,C 0.2369,E1 8.7476,E2 460.1757} C_DIS
LIN {X 131.7622,Y -20.9707,Z 173,A -7.0217,B 8.5873,C 0.2309,E1 8.7485,E2 458.3944} C_DIS
LIN {X 132.3114,Y -17.1604,Z 173,A -5.4674,B 8.5873,C 0.2282,E1 8.749,E2 456.8507} C_DIS
LIN {X 132.7798,Y -13.0532,Z 173,A -3.673,B 8.5875,C 0.2227,E1 8.7496,E2 455.0522} C_DIS
LIN {X 133.1259,Y -8.8729,Z 173,A -2.0138,B 8.5875,C 0.2205,E1 8.7499,E2 453.4089} C_DIS
LIN {X 133.3005,Y -5.6528,Z 173,A -0.5583,B 8.5877,C 0.215,E1 8.7501,E2 451.9434} C_DIS
LIN {X 133.4095,Y -1.7197,Z 173,A 1.0081,B 8.5877,C 0.2127,E1 8.7502,E2 450.3905} C_DIS
LIN {X 133.4013,Y 2.208,Z 173,A 2.7357,B 8.5879,C 0.207,E1 8.7502,E2 448.6563} C_DIS
LIN {X 133.2651,Y 6.423,Z 173,A 4.4751,B 8.588,C 0.2033,E1 8.75,E2 446.9242} C_DIS
LIN {X 133.0385,Y 10.0832,Z 173,A 6.0347,B 8.5881,C 0.1991,E1 8.7497,E2 445.365} C_DIS
LIN {X 132.678,Y 14.0478,Z 173,A 7.7746,B 8.5882,C 0.1935,E1 8.7492,E2 443.62} C_DIS
LIN {X 132.1604,Y 18.2952,Z 173,A 9.6044,B 8.5884,C 0.1884,E1 8.7485,E2 441.7896} C_DIS
LIN {X 131.533,Y 22.3601,Z 173,A 11.3197,B 8.5884,C 0.1844,E1 8.7478,E2 440.0791} C_DIS
LIN {X 130.7767,Y 26.4233,Z 173,A 12.9948,B 8.5885,C 0.1815,E1 8.7469,E2 438.4147} C_DIS
LIN {X 130.0581,Y 29.7592,Z 173,A 14.4663,B 8.5885,C 0.1773,E1 8.746,E2 436.9414} C_DIS
LIN {X 129.1326,Y 33.5565,Z 173,A 16.2409,B 8.5887,C 0.1705,E1 8.7448,E2 435.1537} C_DIS
LIN {X 127.9232,Y 37.9015,Z 173,A 18.3793,B 8.5889,C 0.1609,E1 8.7431,E2 432.9892} C_DIS
LIN {X 126.7974,Y 41.5154,Z 173,A 19.6487,B 8.5889,C 0.164,E1 8.742,E2 431.7622} C_DIS
LIN {X 125.4296,Y 45.4767,Z 173,A 21.9126,B 8.5891,C 0.1493,E1 8.7398,E2 429.4401} C_DIS
LIN {X 123.7973,Y 49.7484,Z 173,A 23.2784,B 8.589,C 0.1567,E1 8.7385,E2 428.1462} C_DIS
LIN {X 122.6404,Y 52.5374,Z 173,A 24.6162,B 8.589,C 0.1524,E1 8.737,E2 426.8025} C_DIS
LIN {X 121.2468,Y 55.6773,Z 173,A 26.0282,B 8.5891,C 0.1498,E1 8.7354,E2 425.3974} C_DIS
LIN {X 119.742,Y 58.8432,Z 173,A 27.5237,B 8.5891,C 0.1462,E1 8.7336,E2 423.9021} C_DIS
LIN {X 118.1877,Y 61.9057,Z 173,A 28.9148,B 8.5892,C 0.1441,E1 8.7318,E2 422.5203} C_DIS
LIN {X 116.2331,Y 65.5062,Z 173,A 30.7852,B 8.5893,C 0.1374,E1 8.7293,E2 420.6355} C_DIS
LIN {X 113.9683,Y 69.3726,Z 173,A 32.7253,B 8.5893,C 0.1323,E1 8.7265,E2 418.6924} C_DIS
LIN {X 111.5994,Y 73.122,Z 173,A 34.5769,B 8.5894,C 0.1288,E1 8.7237,E2 416.8463} C_DIS
LIN {X 108.7948,Y 77.2335,Z 173,A 36.8391,B 8.5896,C 0.1212,E1 8.7201,E2 414.5678} C_DIS
LIN {X 106.1095,Y 80.8825,Z 173,A 39.5526,B 8.5898,C 0.1009,E1 8.7153,E2 411.7594} C_DIS
LIN {X 101.5498,Y 86.538,Z 173,A 41.6458,B 8.5896,C 0.1152,E1 8.7118,E2 409.7906} C_DIS
LIN {X 98.6149,Y 89.8685,Z 173,A 43.5838,B 8.5896,C 0.1105,E1 8.7082,E2 407.8481} C_DIS
LIN {X 96.3916,Y 92.2488,Z 173,A 45.2145,B 8.5898,C 0.1029,E1 8.705,E2 406.1888} C_DIS
LIN {X 93.8142,Y 94.8692,Z 173,A 46.4802,B 8.5898,C 0.106,E1 8.7025,E2 404.9605} C_DIS
LIN {X 90.6105,Y 97.9341,Z 173,A 48.2663,B 8.5898,C 0.1047,E1 8.6989,E2 403.1881} C_DIS
LIN {X 86.9762,Y 101.1747,Z 173,A 50.3937,B 8.5898,C 0.1,E1 8.6945,E2 401.0558} C_DIS
LIN {X 83.7881,Y 103.8302,Z 173,A 52.1933,B 8.5898,C 0.0964,E1 8.6906,E2 399.2537} C_DIS
LIN {X 80.9033,Y 106.0937,Z 173,A 53.9009,B 8.5899,C 0.091,E1 8.6867,E2 397.5297} C_DIS
LIN {X 73.2569,Y 111.5106,Z 173,A 57.7612,B 8.5899,C 0.0877,E1 8.6779,E2 393.6888} C_DIS
LIN {X 69.5176,Y 113.8796,Z 173,A 59.5813,B 8.5899,C 0.0864,E1 8.6736,E2 391.8783} C_DIS
LIN {X 65.9277,Y 115.9946,Z 173,A 61.4142,B 8.59,C 0.083,E1 8.6692,E2 390.04} C_DIS
LIN {X 62.3522,Y 117.9532,Z 173,A 63.0773,B 8.59,C 0.0824,E1 8.6651,E2 388.3874} C_DIS
LIN {X 59.1851,Y 119.5733,Z 173,A 64.5552,B 8.59,C 0.0814,E1 8.6615,E2 386.9153} C_DIS
LIN {X 56.1654,Y 121.0212,Z 173,A 65.9574,B 8.59,C 0.0803,E1 8.6579,E2 385.5176} C_DIS
LIN {X 53.292,Y 122.3141,Z 173,A 67.3817,B 8.59,C 0.0774,E1 8.6543,E2 384.0847} C_DIS
LIN {X 50.0052,Y 123.6938,Z 173,A 68.9356,B 8.59,C 0.0753,E1 8.6502,E2 382.5282} C_DIS
LIN {X 46.2334,Y 125.1539,Z 173,A 70.5897,B 8.59,C 0.0751,E1 8.646,E2 380.8843} C_DIS
LIN {X 41.6189,Y 126.763,Z 173,A 72.8084,B 8.5901,C 0.0709,E1 8.64,E2 378.6514} C_DIS
LIN {X 35.9776,Y 128.4769,Z 173,A 75.6167,B 8.5901,C 0.0637,E1 8.6324,E2 375.8104} C_DIS
LIN {X 32.0807,Y 129.5072,Z 173,A 77.0603,B 8.5901,C 0.0679,E1 8.6286,E2 374.4018} C_DIS
LIN {X 28.1743,Y 130.4106,Z 173,A 78.6462,B 8.5901,C 0.0694,E1 8.6243,E2 372.8326} C_DIS
LIN {X 24.2959,Y 131.1908,Z 173,A 80.4587,B 8.5901,C 0.0664,E1 8.6193,E2 371.0069} C_DIS
LIN {X 20.0601,Y 131.9032,Z 173,A 82.27,B 8.5901,C 0.0662,E1 8.6143,E2 369.2002} C_DIS
LIN {X 15.849,Y 132.4747,Z 173,A 83.9543,B 8.5901,C 0.0681,E1 8.6097,E2 367.5333} C_DIS
LIN {X 12.5876,Y 132.8245,Z 173,A 85.432,B 8.5901,C 0.0665,E1 8.6056,E2 366.0478} C_DIS
LIN {X 8.4198,Y 133.1538,Z 173,A 87.2366,B 8.5901,C 0.066,E1 8.6006,E2 364.2429} C_DIS
LIN {X 4.47,Y 133.3467,Z 173,A 88.9642,B 8.5901,C 0.0653,E1 8.5957,E2 362.5126} C_DIS
LIN {X 0.6245,Y 133.4182,Z 173,A 90.6277,B 8.5901,C 0.065,E1 8.5911,E2 360.8483} C_DIS
LIN {X -3.9498,Y 133.3613,Z 173,A 92.5582,B 8.5901,C 0.0658,E1 8.5857,E2 358.9227} C_DIS
LIN {X -8.1074,Y 133.173,Z 173,A 94.327,B 8.5901,C 0.0664,E1 8.5808,E2 357.1571} C_DIS
LIN {X -11.9787,Y 132.8828,Z 173,A 96.0862,B 8.5901,C 0.0652,E1 8.5759,E2 355.3878} C_DIS
LIN {X -15.849,Y 132.4747,Z 173,A 97.6066,B 8.5901,C 0.0684,E1 8.5717,E2 353.8863} C_DIS
LIN {X -19.1431,Y 132.0392,Z 173,A 99.1552,B 8.5901,C 0.0669,E1 8.5674,E2 352.324} C_DIS
LIN {X -23.3695,Y 131.3568,Z 173,A 100.9577,B 8.5901,C 0.0685,E1 8.5624,E2 350.5269} C_DIS
LIN {X -27.4432,Y 130.5684,Z 173,A 102.8141,B 8.5901,C 0.0682,E1 8.5573,E2 348.6628} C_DIS
LIN {X -31.5084,Y 129.6456,Z 173,A 104.5564,B 8.5901,C 0.0703,E1 8.5526,E2 346.9273} C_DIS
LIN {X -35.7379,Y 128.5439,Z 173,A 106.7509,B 8.5901,C 0.0663,E1 8.5466,E2 344.6961} C_DIS
LIN {X -39.1709,Y 127.5395,Z 173,A 107.897,B 8.5901,C 0.0742,E1 8.5437,E2 343.5976} C_DIS
LIN {X -42.3575,Y 126.517,Z 173,A 109.4169,B 8.5901,C 0.0742,E1 8.5396,E2 342.0689} C_DIS
LIN {X -46.4906,Y 125.0575,Z 173,A 111.183,B 8.5901,C 0.078,E1 8.535,E2 340.3181} C_DIS
LIN {X -52.2156,Y 122.7792,Z 173,A 114.0562,B 8.5901,C 0.0772,E1 8.5275,E2 337.4199} C_DIS
LIN {X -55.777,Y 121.2007,Z 173,A 115.6839,B 8.5901,C 0.0799,E1 8.5234,E2 335.7989} C_DIS
LIN {X -58.4131,Y 119.9542,Z 173,A 117.1466,B 8.5901,C 0.0781,E1 8.5197,E2 334.3122} C_DIS
LIN {X -63.2207,Y 117.4918,Z 173,A 119.2188,B 8.59,C 0.0853,E1 8.5146,E2 332.2714} C_DIS
LIN {X -66.2708,Y 115.7989,Z 173,A 120.7396,B 8.59,C 0.0871,E1 8.5109,E2 330.7492} C_DIS
LIN {X -69.6586,Y 113.7931,Z 173,A 122.4962,B 8.59,C 0.0886,E1 8.5067,E2 328.9861} C_DIS
LIN {X -72.0122,Y 112.3184,Z 173,A 123.8083,B 8.59,C 0.0886,E1 8.5036,E2 327.6609} C_DIS
LIN {X -75.092,Y 110.2837,Z 173,A 125.1564,B 8.5899,C 0.095,E1 8.5005,E2 326.3425} C_DIS
LIN {X -81.257,Y 105.8231,Z 173,A 128.6413,B 8.5899,C 0.0972,E1 8.4926,E2 322.8348} C_DIS
LIN {X -84.7139,Y 103.077,Z 173,A 130.5804,B 8.5899,C 0.1,E1 8.4884,E2 320.8923} C_DIS
LIN {X -88.2939,Y 100.0268,Z 173,A 132.5971,B 8.5898,C 0.1039,E1 8.4841,E2 318.8778} C_DIS
LIN {X -91.633,Y 96.9771,Z 173,A 134.5084,B 8.5898,C 0.1082,E1 8.4802,E2 316.972} C_DIS
LIN {X -94.6688,Y 94.0158,Z 173,A 136.3875,B 8.5897,C 0.1111,E1 8.4765,E2 315.0878} C_DIS
LIN {X -97.0824,Y 91.5214,Z 173,A 137.8982,B 8.5897,C 0.1139,E1 8.4736,E2 313.5762} C_DIS
LIN {X -99.9341,Y 88.3988,Z 173,A 139.7207,B 8.5897,C 0.1178,E1 8.4702,E2 311.7546} C_DIS
LIN {X -102.5816,Y 85.3127,Z 173,A 141.5525,B 8.5896,C 0.1203,E1 8.4669,E2 309.9144} C_DIS
LIN {X -105.4446,Y 81.7472,Z 173,A 143.4518,B 8.5895,C 0.1258,E1 8.4636,E2 308.0247} C_DIS
LIN {X -107.7055,Y 78.7451,Z 173,A 145.0043,B 8.5895,C 0.1306,E1 8.461,E2 306.4812} C_DIS
LIN {X -111.41,Y 73.4097,Z 173,A 147.9702,B 8.5894,C 0.1346,E1 8.4563,E2 303.497} C_DIS
LIN {X -113.1095,Y 70.7638,Z 173,A 149.6508,B 8.5894,C 0.1329,E1 8.4538,E2 301.7782} C_DIS
LIN {X -115.0087,Y 67.6326,Z 173,A 150.9838,B 8.5893,C 0.1405,E1 8.4519,E2 300.4756} C_DIS
LIN {X -117.8105,Y 62.6239,Z 173,A 153.4928,B 8.5892,C 0.1461,E1 8.4486,E2 297.9638} C_DIS
LIN {X -119.5301,Y 59.2728,Z 173,A 155.0657,B 8.5891,C 0.151,E1 8.4466,E2 296.3978} C_DIS
LIN {X -121.0987,Y 55.9978,Z 173,A 156.5757,B 8.5891,C 0.1559,E1 8.4448,E2 294.8953} C_DIS
LIN {X -122.5245,Y 52.8055,Z 173,A 158.1091,B 8.5889,C 0.1594,E1 8.4431,E2 293.3596} C_DIS
LIN {X -123.9921,Y 49.2651,Z 173,A 159.7478,B 8.5889,C 0.164,E1 8.4414,E2 291.7235} C_DIS
LIN {X -125.3226,Y 45.7737,Z 173,A 161.5334,B 8.5889,C 0.1656,E1 8.4396,E2 289.9178} C_DIS
LIN {X -126.6234,Y 42.038,Z 173,A 163.0541,B 8.5887,C 0.173,E1 8.4383,E2 288.4201} C_DIS
LIN {X -127.4335,Y 39.5173,Z 173,A 164.3478,B 8.5887,C 0.1738,E1 8.4372,E2 287.1088} C_DIS
LIN {X -128.499,Y 35.8983,Z 173,A 166.0314,B 8.5886,C 0.1774,E1 8.4359,E2 285.4191} C_DIS
LIN {X -129.6072,Y 31.6677,Z 173,A 167.9582,B 8.5885,C 0.1819,E1 8.4345,E2 283.4883} C_DIS
LIN {X -130.5207,Y 27.6643,Z 173,A 169.6075,B 8.5883,C 0.1886,E1 8.4336,E2 281.8545} C_DIS
LIN {X -131.0274,Y 25.1507,Z 173,A 171.2128,B 8.5884,C 0.1842,E1 8.4327,E2 280.1895} C_DIS
LIN {X -131.7356,Y 21.1425,Z 173,A 172.6431,B 8.5882,C 0.194,E1 8.4321,E2 278.7994} C_DIS
LIN {X -132.2858,Y 17.3551,Z 173,A 174.2192,B 8.5881,C 0.1997,E1 8.4315,E2 277.2329} C_DIS
LIN {X -132.7167,Y 13.6885,Z 173,A 175.9008,B 8.5881,C 0.2029,E1 8.4309,E2 275.5413} C_DIS
LIN {X -133.0656,Y 9.7109,Z 173,A 177.5253,B 8.5879,C 0.2092,E1 8.4306,E2 273.9292} C_DIS
LIN {X -133.2563,Y 6.5985,Z 173,A 178.9653,B 8.5879,C 0.2115,E1 8.4304,E2 272.4783} C_DIS
LIN {X -133.3973,Y 2.4496,Z 173,A -179.188,B 8.5877,C 0.2157,E1 8.4302,E2 270.6255} C_DIS
LIN {X -133.4057,Y -1.9476,Z 173,A -177.2799,B 8.5876,C 0.2209,E1 8.4302,E2 268.7168} C_DIS
LIN {X -133.2827,Y -6.0744,Z 173,A -175.4771,B 8.5875,C 0.2256,E1 8.4304,E2 266.912} C_DIS
LIN {X -133.0605,Y -9.7813,Z 173,A -173.8486,B 8.5874,C 0.2297,E1 8.4307,E2 265.2807} C_DIS
LIN {X -132.6913,Y -13.9248,Z 173,A -172.0121,B 8.5872,C 0.2341,E1 8.4312,E2 263.4397} C_DIS
LIN {X -132.2237,Y -17.829,Z 173,A -170.2221,B 8.5872,C 0.2374,E1 8.4319,E2 261.6389} C_DIS
LIN {X -131.6061,Y -21.9215,Z 173,A -168.5375,B 8.587,C 0.2438,E1 8.4326,E2 259.967} C_DIS
LIN {X -130.2622,Y -28.8616,Z 173,A -165.5834,B 8.5867,C 0.2537,E1 8.4342,E2 257.0253} C_DIS
LIN {X -128.888,Y -34.476,Z 173,A -162.6136,B 8.5867,C 0.2532,E1 8.4363,E2 253.9982} C_DIS
LIN {X -127.9842,Y -37.6932,Z 173,A -161.3941,B 8.5865,C 0.2604,E1 8.4372,E2 252.8061} C_DIS
LIN {X -126.7214,Y -41.7438,Z 173,A -159.5835,B 8.5863,C 0.2656,E1 8.4388,E2 250.9982} C_DIS
LIN {X -125.7305,Y -44.6422,Z 173,A -158.2157,B 8.5863,C 0.2683,E1 8.44,E2 249.625} C_DIS
LIN {X -124.419,Y -48.1725,Z 173,A -156.634,B 8.5861,C 0.2732,E1 8.4416,E2 248.0487} C_DIS
LIN {X -123.1666,Y -51.2899,Z 173,A -155.1168,B 8.5861,C 0.2759,E1 8.4432,E2 246.5234} C_DIS
LIN {X -121.6777,Y -54.7289,Z 173,A -153.5814,B 8.5858,C 0.2812,E1 8.4449,E2 244.998} C_DIS
LIN {X -120.0387,Y -58.2409,Z 173,A -151.7504,B 8.5858,C 0.2829,E1 8.4472,E2 243.1478} C_DIS
LIN {X -118.3979,Y -61.5054,Z 173,A -150.1835,B 8.5856,C 0.2869,E1 8.4492,E2 241.5821} C_DIS
LIN {X -117.0572,Y -64.022,Z 173,A -148.4567,B 8.5858,C 0.2821,E1 8.4516,E2 239.7943} C_DIS
LIN {X -114.7913,Y -68.0019,Z 173,A -146.8807,B 8.5854,C 0.2931,E1 8.4537,E2 238.2675} C_DIS
LIN {X -112.3828,Y -71.9115,Z 173,A -144.934,B 8.5853,C 0.2982,E1 8.4566,E2 236.3249} C_DIS
LIN {X -109.8355,Y -75.7458,Z 173,A -142.8977,B 8.5851,C 0.3019,E1 8.4598,E2 234.2824} C_DIS
LIN {X -107.2315,Y -79.3895,Z 173,A -140.9271,B 8.5851,C 0.3055,E1 8.463,E2 232.3068} C_DIS
LIN {X -104.8475,Y -82.5117,Z 173,A -139.1956,B 8.5849,C 0.3086,E1 8.466,E2 230.5706} C_DIS
LIN {X -101.8461,Y -86.1895,Z 173,A -137.2912,B 8.5847,C 0.3151,E1 8.4694,E2 228.6835} C_DIS
LIN {X -99.2411,Y -89.1763,Z 173,A -135.466,B 8.5847,C 0.3167,E1 8.4728,E2 226.8438} C_DIS
LIN {X -95.9649,Y -92.6926,Z 173,A -133.3708,B 8.5845,C 0.3204,E1 8.4768,E2 224.7455} C_DIS
LIN {X -92.7365,Y -95.9224,Z 173,A -131.4086,B 8.5843,C 0.3242,E1 8.4807,E2 222.7837} C_DIS
LIN {X -89.0569,Y -99.348,Z 173,A -129.1987,B 8.5843,C 0.3274,E1 8.4853,E2 220.5682} C_DIS
LIN {X -85.6593,Y -102.2921,Z 173,A -127.317,B 8.584,C 0.3317,E1 8.4893,E2 218.6929} C_DIS
LIN {X -82.0448,Y -105.2139,Z 173,A -125.207,B 8.584,C 0.3333,E1 8.4939,E2 216.5693} C_DIS
LIN {X -78.6153,Y -107.8005,Z 173,A -123.1706,B 8.584,C 0.3331,E1 8.4986,E2 214.5095} C_DIS
LIN {X -75.9731,Y -109.6783,Z 173,A -121.9995,B 8.5838,C 0.3389,E1 8.5012,E2 213.3658} C_DIS
LIN {X -72.3877,Y -112.0772,Z 173,A -120.1006,B 8.5837,C 0.3409,E1 8.5056,E2 211.4615} C_DIS
LIN {X -68.843,Y -114.2885,Z 173,A -118.3038,B 8.5836,C 0.3434,E1 8.5099,E2 209.6645} C_DIS
LIN {X -65.033,Y -116.4991,Z 173,A -116.3563,B 8.5836,C 0.345,E1 8.5147,E2 207.7101} C_DIS
LIN {X -60.9081,Y -118.7056,Z 173,A -114.5253,B 8.5833,C 0.3505,E1 8.5191,E2 205.9011} C_DIS
LIN {X -57.8236,Y -120.238,Z 173,A -112.9739,B 8.5833,C 0.351,E1 8.523,E2 204.3408} C_DIS
LIN {X -54.6618,Y -121.7077,Z 173,A -111.4641,B 8.5833,C 0.3524,E1 8.5269,E2 202.8294} C_DIS
LIN {X -51.5784,Y -123.0461,Z 173,A -109.9776,B 8.5832,C 0.3532,E1 8.5307,E2 201.3373} C_DIS
LIN {X -47.5179,Y -124.6727,Z 173,A -107.8404,B 8.5833,C 0.3504,E1 8.5364,E2 199.1679} C_DIS
LIN {X -42.5424,Y -126.4554,Z 173,A -105.4649,B 8.5833,C 0.3504,E1 8.5427,E2 196.7788} C_DIS
LIN {X -39.1138,Y -127.557,Z 173,A -103.8548,B 8.5833,C 0.3504,E1 8.547,E2 195.1604} C_DIS
LIN {X -35.1887,Y -128.6975,Z 173,A -102.3753,B 8.5831,C 0.3565,E1 8.5509,E2 193.7151} C_DIS
LIN {X -31.1301,Y -129.7368,Z 173,A -100.7102,B 8.5829,C 0.3599,E1 8.5554,E2 192.0662} C_DIS
LIN {X -27.407,Y -130.5762,Z 173,A -98.9365,B 8.5829,C 0.3583,E1 8.5602,E2 190.2753} C_DIS
LIN {X -23.3267,Y -131.3644,Z 173,A -97.2626,B 8.5829,C 0.3611,E1 8.5648,E2 188.6146} C_DIS
LIN {X -19.2799,Y -132.0197,Z 173,A -95.5106,B 8.5829,C 0.3618,E1 8.5696,E2 186.8632} C_DIS
LIN {X -16.1185,Y -132.4426,Z 173,A -94.0949,B 8.5829,C 0.3613,E1 8.5736,E2 185.4413} C_DIS
LIN {X -12.2369,Y -132.8581,Z 173,A -92.4629,B 8.5829,C 0.3624,E1 8.5781,E2 183.8142} C_DIS
LIN {X -8.4456,Y -133.1522,Z 173,A -90.8098,B 8.5829,C 0.3621,E1 8.5827,E2 182.1578} C_DIS
LIN {X -4.6087,Y -133.3413,Z 173,A -89.0008,B 8.5829,C 0.3592,E1 8.5878,E2 180.3284} C_DIS
LIN {X 0.2699,Y -133.4202,Z 173,A -87.0497,B 8.5829,C 0.3617,E1 8.5932,E2 178.3943} C_DIS
LIN {X 0.2699,Y -133.4202,Z 173,A -87.0497,B 8.5829,C 0.3617,E1 8.5932,E2 178.3943} C_DIS
Enddeposition()
LIN {X 0.9731,Y -134.3248,Z 173,A -87.1741,B 8.5823,C 0.3746,E1 8.5926,E2 178.6052} C_DIS
Startdeposition()
$VEL.CP = VEL_PRINT
LIN {X -3.2114,Y -134.2904,Z 173,A -89.5409,B 8.5818,C 0.3855,E1 8.5858,E2 181.045} C_DIS
LIN {X -6.6867,Y -134.1616,Z 173,A -90.6707,B 8.5821,C 0.379,E1 8.5828,E2 182.1317} C_DIS
LIN {X -10.4705,Y -133.9211,Z 173,A -92.3613,B 8.5821,C 0.3802,E1 8.578,E2 183.8321} C_DIS
LIN {X -14.297,Y -133.565,Z 173,A -94.1396,B 8.5819,C 0.3824,E1 8.5731,E2 185.6281} C_DIS
LIN {X -18.9289,Y -132.9876,Z 173,A -95.9265,B 8.5821,C 0.3782,E1 8.5682,E2 187.3906} C_DIS
LIN {X -22.2357,Y -132.4748,Z 173,A -97.3669,B 8.5821,C 0.378,E1 8.5642,E2 188.8329} C_DIS
LIN {X -26.2247,Y -131.7443,Z 173,A -99.1372,B 8.5821,C 0.378,E1 8.5593,E2 190.6089} C_DIS
LIN {X -29.715,Y -131.0001,Z 173,A -100.6583,B 8.5821,C 0.3772,E1 8.5552,E2 192.1302} C_DIS
LIN {X -33.1386,Y -130.176,Z 173,A -102.1177,B 8.5823,C 0.3756,E1 8.5512,E2 193.5846} C_DIS
LIN {X -36.0112,Y -129.4108,Z 173,A -103.3646,B 8.5823,C 0.3744,E1 8.5479,E2 194.8292} C_DIS
LIN {X -40.8762,Y -127.9573,Z 173,A -106.0427,B 8.582,C 0.3817,E1 8.5406,E2 197.5708} C_DIS
LIN {X -44.9057,Y -126.6013,Z 173,A -107.3401,B 8.5824,C 0.3713,E1 8.5373,E2 198.805} C_DIS
LIN {X -49.3047,Y -124.9537,Z 173,A -109.5436,B 8.5824,C 0.3729,E1 8.5315,E2 201.0335} C_DIS
LIN {X -53.7046,Y -123.1255,Z 173,A -111.5774,B 8.5824,C 0.3708,E1 8.5263,E2 203.0675} C_DIS
LIN {X -57.5449,Y -121.3781,Z 173,A -113.2806,B 8.5826,C 0.3672,E1 8.522,E2 204.7589} C_DIS
LIN {X -60.6725,Y -119.845,Z 173,A -114.7668,B 8.5826,C 0.3654,E1 8.5183,E2 206.2452} C_DIS
LIN {X -63.8709,Y -118.1738,Z 173,A -116.4292,B 8.5826,C 0.3656,E1 8.5141,E2 207.9228} C_DIS
LIN {X -67.7049,Y -116.0199,Z 173,A -118.3408,B 8.5828,C 0.3637,E1 8.5095,E2 209.8388} C_DIS
LIN {X -71.48,Y -113.7326,Z 173,A -120.2199,B 8.5828,C 0.3609,E1 8.505,E2 211.7172} C_DIS
LIN {X -75.2737,Y -111.2578,Z 173,A -122.1085,B 8.583,C 0.3573,E1 8.5006,E2 213.6002} C_DIS
LIN {X -81.4864,Y -106.7914,Z 173,A -125.128,B 8.5834,C 0.348,E1 8.4939,E2 216.5893} C_DIS
LIN {X -85.4017,Y -103.6875,Z 173,A -127.6377,B 8.5834,C 0.3506,E1 8.4883,E2 219.1452} C_DIS
LIN {X -88.9109,Y -100.694,Z 173,A -129.5763,B 8.5834,C 0.3465,E1 8.4842,E2 221.0797} C_DIS
LIN {X -92.2387,Y -97.6548,Z 173,A -131.4826,B 8.5836,C 0.3426,E1 8.4803,E2 222.9835} C_DIS
LIN {X -95.2151,Y -94.7551,Z 173,A -133.3193,B 8.5837,C 0.3402,E1 8.4767,E2 224.8275} C_DIS
LIN {X -97.2882,Y -92.6256,Z 173,A -134.9599,B 8.5836,C 0.3436,E1 8.4734,E2 226.5133} C_DIS
LIN {X -99.998,Y -89.693,Z 173,A -136.4329,B 8.5839,C 0.3364,E1 8.4707,E2 227.9576} C_DIS
LIN {X -103.229,Y -85.9555,Z 173,A -138.4641,B 8.5841,C 0.3307,E1 8.4671,E2 229.9787} C_DIS
LIN {X -105.2856,Y -83.4233,Z 173,A -140.1619,B 8.5841,C 0.3325,E1 8.4641,E2 231.7132} C_DIS
LIN {X -107.525,Y -80.5167,Z 173,A -141.4992,B 8.5843,C 0.3254,E1 8.4619,E2 233.0222} C_DIS
LIN {X -110.1844,Y -76.8366,Z 173,A -143.7514,B 8.5843,C 0.3258,E1 8.4582,E2 235.3118} C_DIS
LIN {X -112.3552,Y -73.6262,Z 173,A -145.0669,B 8.5846,C 0.3167,E1 8.4562,E2 236.5854} C_DIS
LIN {X -114.6881,Y -69.9371,Z 173,A -146.9867,B 8.5847,C 0.3131,E1 8.4534,E2 238.5114} C_DIS
LIN {X -119.9385,Y -60.4888,Z 173,A -152.215,B 8.5848,C 0.311,E1 8.4464,E2 243.8117} C_DIS
LIN {X -122.0878,Y -56.0233,Z 173,A -153.8361,B 8.5853,C 0.2981,E1 8.4445,E2 245.372} C_DIS
LIN {X -123.7958,Y -52.1408,Z 173,A -155.5813,B 8.5855,C 0.2923,E1 8.4426,E2 247.1081} C_DIS
LIN {X -125.1662,Y -48.758,Z 173,A -157.2178,B 8.5855,C 0.2894,E1 8.4409,E2 248.7533} C_DIS
LIN {X -126.6211,Y -44.8506,Z 173,A -159.0923,B 8.5857,C 0.2861,E1 8.4391,E2 250.6383} C_DIS
LIN {X -128.0412,Y -40.6134,Z 173,A -161.445,B 8.5857,C 0.2876,E1 8.437,E2 253.0433} C_DIS
LIN {X -129.3385,Y -36.2699,Z 173,A -162.6752,B 8.5861,C 0.2717,E1 8.4362,E2 254.1872} C_DIS
LIN {X -130.0567,Y -33.6071,Z 173,A -164.5413,B 8.5859,C 0.2788,E1 8.4348,E2 256.1357} C_DIS
LIN {X -131.0411,Y -29.5356,Z 173,A -165.8781,B 8.5863,C 0.2671,E1 8.434,E2 257.4169} C_DIS
LIN {X -131.8925,Y -25.4636,Z 173,A -167.8098,B 8.5863,C 0.2644,E1 8.4329,E2 259.3662} C_DIS
LIN {X -132.7133,Y -20.766,Z 173,A -169.7728,B 8.5866,C 0.2576,E1 8.432,E2 261.319} C_DIS
LIN {X -133.2826,Y -16.741,Z 173,A -171.6075,B 8.5866,C 0.2541,E1 8.4313,E2 263.1645} C_DIS
LIN {X -133.7015,Y -12.9591,Z 173,A -173.2095,B 8.5868,C 0.2491,E1 8.4309,E2 264.7624} C_DIS
LIN {X -134.0495,Y -8.6557,Z 173,A -175.0958,B 8.5869,C 0.2445,E1 8.4305,E2 266.6526} C_DIS
LIN {X -134.2399,Y -4.8807,Z 173,A -176.7797,B 8.5871,C 0.2409,E1 8.4303,E2 268.3436} C_DIS
LIN {X -134.3286,Y -0.509,Z 173,A -178.603,B 8.5872,C 0.2349,E1 8.4303,E2 270.1603} C_DIS
LIN {X -134.2864,Y 3.369,Z 173,A 179.7031,B 8.5873,C 0.2307,E1 8.4303,E2 271.8574} C_DIS
LIN {X -134.1487,Y 6.9434,Z 173,A 178.1651,B 8.5874,C 0.2265,E1 8.4305,E2 273.3955} C_DIS
LIN {X -133.8668,Y 11.1231,Z 173,A 176.3864,B 8.5876,C 0.2212,E1 8.4308,E2 275.1714} C_DIS
LIN {X -133.513,Y 14.7798,Z 173,A 174.7299,B 8.5876,C 0.218,E1 8.4313,E2 276.8372} C_DIS
LIN {X -132.9964,Y 18.8672,Z 173,A 172.975,B 8.5878,C 0.2129,E1 8.432,E2 278.5901} C_DIS
LIN {X -132.4119,Y 22.6125,Z 173,A 171.0427,B 8.5878,C 0.2129,E1 8.4329,E2 280.5586} C_DIS
LIN {X -131.8195,Y 25.8456,Z 173,A 169.7739,B 8.5879,C 0.207,E1 8.4335,E2 281.8102} C_DIS
LIN {X -131.0208,Y 29.6243,Z 173,A 168.1851,B 8.5881,C 0.2014,E1 8.4345,E2 283.3904} C_DIS
LIN {X -129.9114,Y 34.1642,Z 173,A 166.2293,B 8.5882,C 0.1952,E1 8.4358,E2 285.3396} C_DIS
LIN {X -129.0492,Y 37.2889,Z 173,A 164.7765,B 8.5882,C 0.1924,E1 8.4369,E2 286.7994} C_DIS
LIN {X -128.1287,Y 40.3398,Z 173,A 163.3865,B 8.5883,C 0.1891,E1 8.4381,E2 288.1919} C_DIS
LIN {X -126.7424,Y 44.5037,Z 173,A 160.8967,B 8.5883,C 0.1931,E1 8.4404,E2 290.7532} C_DIS
LIN {X -125.0354,Y 49.0944,Z 173,A 159.2539,B 8.5885,C 0.1808,E1 8.442,E2 292.3409} C_DIS
LIN {X -123.4262,Y 53.0093,Z 173,A 157.6496,B 8.5887,C 0.173,E1 8.4437,E2 293.9193} C_DIS
LIN {X -122.2473,Y 55.6785,Z 173,A 156.1805,B 8.5887,C 0.173,E1 8.4454,E2 295.4141} C_DIS
LIN {X -120.6172,Y 59.1228,Z 173,A 154.6751,B 8.5887,C 0.1669,E1 8.4472,E2 296.9035} C_DIS
LIN {X -118.6848,Y 62.9132,Z 173,A 152.4527,B 8.5887,C 0.1684,E1 8.4502,E2 299.1725} C_DIS
LIN {X -116.9741,Y 66.0412,Z 173,A 151.1901,B 8.5889,C 0.1606,E1 8.4518,E2 300.403} C_DIS
LIN {X -114.0863,Y 70.9138,Z 173,A 148.7214,B 8.589,C 0.1554,E1 8.4554,E2 302.8755} C_DIS
LIN {X -112.0644,Y 74.068,Z 173,A 146.9862,B 8.589,C 0.1536,E1 8.4581,E2 304.6254} C_DIS
LIN {X -108.8513,Y 78.7136,Z 173,A 144.6371,B 8.5892,C 0.1469,E1 8.4618,E2 306.9649} C_DIS
LIN {X -106.1677,Y 82.2973,Z 173,A 142.7262,B 8.5892,C 0.1425,E1 8.4651,E2 308.874} C_DIS
LIN {X -103.6923,Y 85.3959,Z 173,A 140.9094,B 8.5892,C 0.1406,E1 8.4683,E2 310.7041} C_DIS
LIN {X -100.4895,Y 89.1423,Z 173,A 138.9645,B 8.5894,C 0.1335,E1 8.4718,E2 312.6283} C_DIS
LIN {X -97.2774,Y 92.6368,Z 173,A 136.8039,B 8.5894,C 0.1313,E1 8.4759,E2 314.803} C_DIS
LIN {X -94.7556,Y 95.2146,Z 173,A 135.1539,B 8.5894,C 0.1298,E1 8.4792,E2 316.4648} C_DIS
LIN {X -91.178,Y 98.6465,Z 173,A 133.2261,B 8.5895,C 0.1227,E1 8.4831,E2 318.3684} C_DIS
LIN {X -87.2099,Y 102.1711,Z 173,A 130.8205,B 8.5895,C 0.1205,E1 8.4882,E2 320.7888} C_DIS
LIN {X -83.8972,Y 104.9084,Z 173,A 128.9581,B 8.5896,C 0.1176,E1 8.4922,E2 322.653} C_DIS
LIN {X -81.6316,Y 106.6804,Z 173,A 127.2703,B 8.5896,C 0.1227,E1 8.4961,E2 324.394} C_DIS
LIN {X -77.9468,Y 109.4019,Z 173,A 125.5879,B 8.5896,C 0.1151,E1 8.4998,E2 326.0427} C_DIS
LIN {X -73.5697,Y 112.3924,Z 173,A 123.6027,B 8.5897,C 0.107,E1 8.5043,E2 327.9933} C_DIS
LIN {X -69.7781,Y 114.7848,Z 173,A 121.5208,B 8.5897,C 0.1068,E1 8.5093,E2 330.0936} C_DIS
LIN {X -66.154,Y 116.9111,Z 173,A 119.7376,B 8.5897,C 0.104,E1 8.5136,E2 331.8743} C_DIS
LIN {X -62.4113,Y 118.9484,Z 173,A 117.3361,B 8.5897,C 0.1109,E1 8.5197,E2 334.343} C_DIS
LIN {X -57.8288,Y 121.2424,Z 173,A 115.793,B 8.5899,C 0.0977,E1 8.5234,E2 335.8086} C_DIS
LIN {X -54.6156,Y 122.7237,Z 173,A 114.2239,B 8.5899,C 0.0968,E1 8.5274,E2 337.3837} C_DIS
LIN {X -51.4283,Y 124.0934,Z 173,A 112.8106,B 8.5899,C 0.094,E1 8.531,E2 338.788} C_DIS
LIN {X -42.9339,Y 127.2827,Z 173,A 109.0126,B 8.5899,C 0.0889,E1 8.541,E2 342.5747} C_DIS
LIN {X -35.2896,Y 129.6113,Z 173,A 105.3438,B 8.5899,C 0.0905,E1 8.5509,E2 346.2722} C_DIS
LIN {X -31.6986,Y 130.5343,Z 173,A 103.8691,B 8.5899,C 0.0875,E1 8.5548,E2 347.7331} C_DIS
LIN {X -28.0243,Y 131.3724,Z 173,A 102.2043,B 8.5899,C 0.0875,E1 8.5594,E2 349.4038} C_DIS
LIN {X -23.9409,Y 132.1775,Z 173,A 100.5022,B 8.5899,C 0.0852,E1 8.564,E2 351.0961} C_DIS
LIN {X -20.8204,Y 132.7048,Z 173,A 99.1176,B 8.5899,C 0.0852,E1 8.5678,E2 352.484} C_DIS
LIN {X -17.5219,Y 133.1803,Z 173,A 97.7318,B 8.5899,C 0.0839,E1 8.5716,E2 353.8647} C_DIS
LIN {X -13.9987,Y 133.5971,Z 173,A 96.0577,B 8.5899,C 0.0862,E1 8.5763,E2 355.5571} C_DIS
LIN {X -9.6521,Y 133.9809,Z 173,A 94.2716,B 8.5899,C 0.0844,E1 8.5813,E2 357.3333} C_DIS
LIN {X -5.485,Y 134.2163,Z 173,A 92.4889,B 8.5899,C 0.0842,E1 8.5863,E2 359.1154} C_DIS
LIN {X -1.486,Y 134.322,Z 173,A 90.6713,B 8.5899,C 0.0861,E1 8.5914,E2 360.9455} C_DIS
LIN {X 3.2279,Y 134.2903,Z 173,A 88.7504,B 8.5899,C 0.0845,E1 8.5967,E2 362.8548} C_DIS
LIN {X 7.2521,Y 134.1331,Z 173,A 87.0307,B 8.5899,C 0.0848,E1 8.6015,E2 364.5741} C_DIS
LIN {X 11.2431,Y 133.8567,Z 173,A 85.4396,B 8.59,C 0.083,E1 8.6059,E2 366.1507} C_DIS
LIN {X 14.9044,Y 133.4996,Z 173,A 83.8251,B 8.59,C 0.0843,E1 8.6104,E2 367.7701} C_DIS
LIN {X 18.5302,Y 133.0446,Z 173,A 82.2551,B 8.59,C 0.0851,E1 8.6147,E2 369.341} C_DIS
LIN {X 21.9718,Y 132.5188,Z 173,A 80.8043,B 8.59,C 0.0851,E1 8.6187,E2 370.7872} C_DIS
LIN {X 25.4849,Y 131.8885,Z 173,A 79.2808,B 8.59,C 0.0859,E1 8.6229,E2 372.3104} C_DIS
LIN {X 29.4528,Y 131.06,Z 173,A 77.4959,B 8.59,C 0.0879,E1 8.6278,E2 374.1015} C_DIS
LIN {X 32.9458,Y 130.2249,Z 173,A 76.1276,B 8.59,C 0.0859,E1 8.6315,E2 375.45} C_DIS
LIN {X 35.2691,Y 129.6167,Z 173,A 74.8341,B 8.59,C 0.0917,E1 8.635,E2 376.7753} C_DIS
LIN {X 41.8042,Y 127.6588,Z 173,A 72.1055,B 8.59,C 0.0907,E1 8.6423,E2 379.4819} C_DIS
LIN {X 46.3065,Y 126.096,Z 173,A 69.9441,B 8.5899,C 0.0951,E1 8.648,E2 381.6584} C_DIS
LIN {X 51.1296,Y 124.2181,Z 173,A 67.841,B 8.5899,C 0.0954,E1 8.6534,E2 383.7488} C_DIS
LIN {X 54.5632,Y 122.7471,Z 173,A 66.3001,B 8.5899,C 0.0962,E1 8.6573,E2 385.2833} C_DIS
LIN {X 57.6641,Y 121.3211,Z 173,A 64.8657,B 8.5899,C 0.0976,E1 8.661,E2 386.7152} C_DIS
LIN {X 60.7022,Y 119.8299,Z 173,A 63.4384,B 8.5899,C 0.0991,E1 8.6645,E2 388.1405} C_DIS
LIN {X 63.985,Y 118.1123,Z 173,A 61.7661,B 8.5898,C 0.103,E1 8.6687,E2 389.824} C_DIS
LIN {X 67.7381,Y 116.0004,Z 173,A 59.948,B 8.5898,C 0.1053,E1 8.6731,E2 391.6399} C_DIS
LIN {X 71.4438,Y 113.7554,Z 173,A 58.1109,B 8.5898,C 0.1078,E1 8.6774,E2 393.4759} C_DIS
LIN {X 75.6194,Y 111.0228,Z 173,A 55.8092,B 8.5896,C 0.1146,E1 8.6828,E2 395.7984} C_DIS
LIN {X 78.3385,Y 109.1218,Z 173,A 54.6148,B 8.5896,C 0.1126,E1 8.6855,E2 396.9668} C_DIS
LIN {X 81.4202,Y 106.842,Z 173,A 52.9744,B 8.5896,C 0.1155,E1 8.6891,E2 398.6081} C_DIS
LIN {X 84.9951,Y 104.0205,Z 173,A 51.0834,B 8.5896,C 0.118,E1 8.6932,E2 400.4933} C_DIS
LIN {X 88.2157,Y 101.3037,Z 173,A 49.5173,B 8.5896,C 0.1167,E1 8.6965,E2 402.032} C_DIS
LIN {X 90.8376,Y 98.9594,Z 173,A 47.807,B 8.5896,C 0.1238,E1 8.7001,E2 403.768} C_DIS
LIN {X 94.2146,Y 95.7501,Z 173,A 45.9025,B 8.5895,C 0.1261,E1 8.7039,E2 405.6632} C_DIS
LIN {X 97.4172,Y 92.4905,Z 173,A 43.8816,B 8.5895,C 0.1316,E1 8.7079,E2 407.6935} C_DIS
Enddeposition()
END
